					// If this exact part has not yet been actuated, an edge behind the
					// final array of the still-airborne previous part is its duplicate,
					// not permission to advance the next queue sequence.
					IF BatchSensorOrderInvalid
						AND NOT BatchCanResyncSkippedSensors
						AND (BatchNextSensorSequence[BatchLoopIndex] > 1) THEN
						BatchPreviousSlotIndex := UDINT_TO_INT(
							(BatchNextSensorSequence[BatchLoopIndex] - 2) MOD 128);
						IF (BatchQueueArrayMask[BatchPreviousSlotIndex] AND BYTE#8) <> BYTE#0 THEN
							BatchPreviousLastRequiredSensor := 8;
							BatchPreviousLastRequiredArrayMask := BYTE#8;
						ELSIF (BatchQueueArrayMask[BatchPreviousSlotIndex] AND BYTE#4) <> BYTE#0 THEN
							BatchPreviousLastRequiredSensor := 6;
							BatchPreviousLastRequiredArrayMask := BYTE#4;
						ELSIF (BatchQueueArrayMask[BatchPreviousSlotIndex] AND BYTE#2) <> BYTE#0 THEN
							BatchPreviousLastRequiredSensor := 4;
							BatchPreviousLastRequiredArrayMask := BYTE#2;
						ELSIF (BatchQueueArrayMask[BatchPreviousSlotIndex] AND BYTE#1) <> BYTE#0 THEN
							BatchPreviousLastRequiredSensor := 2;
							BatchPreviousLastRequiredArrayMask := BYTE#1;
						END_IF
						BatchIgnoreAirborneDuplicate :=
							(BatchQueueSequence[BatchPreviousSlotIndex]
								= (BatchNextSensorSequence[BatchLoopIndex] - 1))
							AND NOT BatchQueueExitSeen[BatchPreviousSlotIndex]
							AND (BatchPreviousLastRequiredArrayMask <> BYTE#0)
							AND ((BatchQueueActuatedMask[BatchPreviousSlotIndex]
								AND BatchPreviousLastRequiredArrayMask) <> BYTE#0)
							AND (BatchLoopIndex > BatchPreviousLastRequiredSensor);
					END_IF
				END_IF
				ReorientationFaultQueueSlotSequence := BatchQueueSequence[BatchSlotIndex];
				IF (BatchNextSensorSequence[BatchLoopIndex] > ReorientationQueueEnqueueAck)
					OR (BatchQueueSequence[BatchSlotIndex] <> BatchNextSensorSequence[BatchLoopIndex]) THEN
					ReorientationFaultDetail := 2;
					ReorientationWarningCode := 4;
					ReorientationWarningSensor := INT_TO_UINT(BatchLoopIndex);
					ReorientationWarningSequence := BatchNextSensorSequence[BatchLoopIndex];
					ReorientationWarningPreviousSequence := ReorientationFaultPreviousSequence;
					ReorientationWarningSkippedBarrierMask := BYTE#0;
					ReorientationWarningCounter := ReorientationWarningCounter + 1;
					IF (BatchLoopIndex MOD 2) = 1 THEN
						BatchJobIndex := (BatchLoopIndex + 1) / 2;
						PairedFirstBarrierLocked[BatchJobIndex] := TRUE;
						PairedFirstBarrierLockStartMs[BatchJobIndex] := LightBarrierEventClockMs;
						PairedSecondBarrierLocked[BatchJobIndex] := FALSE;
					ELSE
						BatchJobIndex := BatchLoopIndex / 2;
						PairedSecondBarrierLocked[BatchJobIndex] := TRUE;
						PairedSecondBarrierLockStartMs[BatchJobIndex] := LightBarrierEventClockMs;
						PairedFirstBarrierLocked[BatchJobIndex] := FALSE;
					END_IF
				ELSIF BatchIgnoreAirborneDuplicate THEN
					// The partner gate admitted another optical edge from the already
					// actuated previous part. Keep the current cursor unchanged and
					// restart this sensor's inhibit instead of faulting or misassigning it.
					ReorientationWarningCode := 2;
					ReorientationWarningSensor := INT_TO_UINT(BatchLoopIndex);
					ReorientationWarningSequence := BatchNextSensorSequence[BatchLoopIndex];
					ReorientationWarningPreviousSequence :=
						BatchNextSensorSequence[BatchLoopIndex] - 1;
					ReorientationWarningSkippedBarrierMask := BYTE#0;
					ReorientationWarningCounter := ReorientationWarningCounter + 1;
					IF (BatchLoopIndex MOD 2) = 1 THEN
						BatchJobIndex := (BatchLoopIndex + 1) / 2;
						PairedFirstBarrierLocked[BatchJobIndex] := TRUE;
						PairedFirstBarrierLockStartMs[BatchJobIndex] := LightBarrierEventClockMs;
						PairedSecondBarrierLocked[BatchJobIndex] := FALSE;
					ELSE
						BatchJobIndex := BatchLoopIndex / 2;
						PairedSecondBarrierLocked[BatchJobIndex] := TRUE;
						PairedSecondBarrierLockStartMs[BatchJobIndex] := LightBarrierEventClockMs;
						PairedFirstBarrierLocked[BatchJobIndex] := FALSE;
					END_IF
				ELSIF BatchSensorOrderInvalid AND NOT BatchCanResyncSkippedSensors THEN
					ReorientationFaultDetail := 3;
					ReorientationWarningCode := 5;
					ReorientationWarningSensor := INT_TO_UINT(BatchLoopIndex);
					ReorientationWarningSequence := BatchNextSensorSequence[BatchLoopIndex];
					ReorientationWarningPreviousSequence := ReorientationFaultPreviousSequence;
					ReorientationWarningSkippedBarrierMask := BYTE#0;
					ReorientationWarningCounter := ReorientationWarningCounter + 1;
					IF (BatchLoopIndex MOD 2) = 1 THEN
						BatchJobIndex := (BatchLoopIndex + 1) / 2;
						PairedFirstBarrierLocked[BatchJobIndex] := TRUE;
						PairedFirstBarrierLockStartMs[BatchJobIndex] := LightBarrierEventClockMs;
						PairedSecondBarrierLocked[BatchJobIndex] := FALSE;
					ELSE
						BatchJobIndex := BatchLoopIndex / 2;
						PairedSecondBarrierLocked[BatchJobIndex] := TRUE;
						PairedSecondBarrierLockStartMs[BatchJobIndex] := LightBarrierEventClockMs;
						PairedFirstBarrierLocked[BatchJobIndex] := FALSE;
					END_IF
				ELSE
					IF BatchCanResyncSkippedSensors THEN
						BatchSkippedBarrierMask := BYTE#0;
						FOR BatchResyncIndex := BatchLastRequiredSensor + 1 TO BatchLoopIndex - 1 DO
							IF BatchSensorSequence[BatchResyncIndex]
								< BatchNextSensorSequence[BatchLoopIndex] THEN
								BatchSensorSequence[BatchResyncIndex] :=
									BatchNextSensorSequence[BatchLoopIndex];
								BatchNextSensorSequence[BatchResyncIndex] :=
									BatchNextSensorSequence[BatchLoopIndex] + 1;
								BatchSensorNeedsClear[BatchResyncIndex] := FALSE;
								BatchSkippedBarrierMask := BatchSkippedBarrierMask
									OR SHL(BYTE#1, BatchResyncIndex - 1);
								// Advance the alternating pair gate just as the virtual sensor
								// acceptance advances its sequence cursor.
								IF (BatchResyncIndex MOD 2) = 1 THEN
									BatchJobIndex := (BatchResyncIndex + 1) / 2;
									PairedFirstBarrierLocked[BatchJobIndex] := TRUE;
									PairedFirstBarrierLockStartMs[BatchJobIndex] := LightBarrierEventClockMs;
									PairedSecondBarrierLocked[BatchJobIndex] := FALSE;
								ELSE
									BatchJobIndex := BatchResyncIndex / 2;
									PairedSecondBarrierLocked[BatchJobIndex] := TRUE;
									PairedSecondBarrierLockStartMs[BatchJobIndex] := LightBarrierEventClockMs;
									PairedFirstBarrierLocked[BatchJobIndex] := FALSE;
								END_IF
							END_IF
						END_FOR
						// The physical current edge was evaluated before the virtual ones;
						// re-apply it last so a skipped odd sensor in the same pair cannot
						// overwrite the correct final gate phase.
						IF (BatchLoopIndex MOD 2) = 1 THEN
							BatchJobIndex := (BatchLoopIndex + 1) / 2;
							PairedFirstBarrierLocked[BatchJobIndex] := TRUE;
							PairedFirstBarrierLockStartMs[BatchJobIndex] := LightBarrierEventClockMs;
							PairedSecondBarrierLocked[BatchJobIndex] := FALSE;
						ELSE
							BatchJobIndex := BatchLoopIndex / 2;
							PairedSecondBarrierLocked[BatchJobIndex] := TRUE;
							PairedSecondBarrierLockStartMs[BatchJobIndex] := LightBarrierEventClockMs;
							PairedFirstBarrierLocked[BatchJobIndex] := FALSE;
						END_IF
						ReorientationWarningCode := 1;
						ReorientationWarningSensor := INT_TO_UINT(BatchLoopIndex);
						ReorientationWarningSequence := BatchNextSensorSequence[BatchLoopIndex];
						ReorientationWarningPreviousSequence := ReorientationFaultPreviousSequence;
						ReorientationWarningSkippedBarrierMask := BatchSkippedBarrierMask;
						ReorientationWarningCounter := ReorientationWarningCounter + 1;
					END_IF
					BatchSensorSequence[BatchLoopIndex] := BatchNextSensorSequence[BatchLoopIndex];
					IF (BatchLoopIndex MOD 2) = 1 THEN
						BatchJobIndex := (BatchLoopIndex + 1) / 2;
						BatchQueuePairStartMs[BatchSlotIndex, BatchJobIndex] := LightBarrierEventClockMs;
						IF BatchLoopIndex = 1 THEN
							ReorientationQueueEnteredCount := ReorientationQueueEnteredCount + 1;
						END_IF
					ELSE
						BatchJobIndex := BatchLoopIndex / 2;
						IF (BatchQueueArrayMask[BatchSlotIndex] AND SHL(BYTE#1, BatchJobIndex - 1)) <> BYTE#0 THEN
							IF BatchJobCount[BatchJobIndex] >= 16 THEN
								ReorientationFaultCode := 95; // per-array job FIFO overflow
								ReorientationState := 95;
								ReorientationSafeLatch := TRUE;
							ELSE
								BatchElapsedMs := LightBarrierEventClockMs - BatchQueuePairStartMs[BatchSlotIndex, BatchJobIndex];
								BatchNozzleCount := 0;
								FOR BatchSlotIndex := 0 TO 5 DO
									IF (BatchQueueNozzleMask[UDINT_TO_INT((BatchNextSensorSequence[BatchLoopIndex] - 1) MOD 128), BatchJobIndex]
										AND SHL(BYTE#1, BatchSlotIndex)) <> BYTE#0 THEN
										BatchNozzleCount := BatchNozzleCount + 1;
									END_IF
								END_FOR
								BatchSlotIndex := UDINT_TO_INT((BatchNextSensorSequence[BatchLoopIndex] - 1) MOD 128);
				// One response-delay setting is used for every nozzle count.
				BatchResponseDelayMs := BatchQueueForceSingleMs[BatchSlotIndex, BatchJobIndex];
				BatchComputedDelayMs := UINT_TO_REAL(BatchQueueDelayMs[BatchSlotIndex, BatchJobIndex]);
				IF (BatchElapsedMs > 0) AND (BatchPairSpacingMm[BatchJobIndex] > 0.0)
					AND ((BatchSensorToArraySpacingMm[BatchJobIndex]
					+ BatchQueueOffsetMm[BatchSlotIndex, BatchJobIndex]) > 0.0) THEN
					BatchComputedDelayMs := BatchComputedDelayMs
						+ (BatchSensorToArraySpacingMm[BatchJobIndex]
						+ BatchQueueOffsetMm[BatchSlotIndex, BatchJobIndex])
						* UDINT_TO_REAL(BatchElapsedMs) / BatchPairSpacingMm[BatchJobIndex]
						- BatchResponseDelayMs;
								END_IF
								IF BatchComputedDelayMs < 0.0 THEN BatchComputedDelayMs := 0.0; END_IF
								IF BatchComputedDelayMs > 31000.0 THEN BatchComputedDelayMs := 31000.0; END_IF
								BatchJobSequence[BatchJobTail[BatchJobIndex], BatchJobIndex] := BatchQueueSequence[BatchSlotIndex];
								BatchJobNozzleMask[BatchJobTail[BatchJobIndex], BatchJobIndex] := BatchQueueNozzleMask[BatchSlotIndex, BatchJobIndex];
								BatchJobPressureMbar[BatchJobTail[BatchJobIndex], BatchJobIndex] := BatchQueuePressureMbar[BatchSlotIndex, BatchJobIndex];
								BatchJobDelayCycles[BatchJobTail[BatchJobIndex], BatchJobIndex] := REAL_TO_INT(BatchComputedDelayMs);
								BatchJobPulseCycles[BatchJobTail[BatchJobIndex], BatchJobIndex] := UINT_TO_INT(BatchQueuePulseMs[BatchSlotIndex, BatchJobIndex]);
								BatchJobTail[BatchJobIndex] := (BatchJobTail[BatchJobIndex] + 1) MOD 16;
								BatchJobCount[BatchJobIndex] := BatchJobCount[BatchJobIndex] + 1;
								BatchQueueTriggeredMask[BatchSlotIndex] := BatchQueueTriggeredMask[BatchSlotIndex]
									OR SHL(BYTE#1, BatchJobIndex - 1);
							END_IF
						END_IF
						IF BatchLoopIndex = 8 THEN
							BatchQueueExitSeen[BatchSlotIndex] := TRUE;
							ReorientationExitSeen := TRUE;
						END_IF
					END_IF
					BatchNextSensorSequence[BatchLoopIndex] := BatchNextSensorSequence[BatchLoopIndex] + 1;
				END_IF
			END_IF
		END_IF
		// Preserve the first faulting sensor and its context. Without EXIT, a
		// second edge in this same 1-ms scan could overwrite the diagnostics.
		IF ReorientationSafeLatch THEN
			EXIT;
		END_IF
	END_FOR
END_IF

ReorientationSensorSequence1 := BatchSensorSequence[1];
ReorientationSensorSequence2 := BatchSensorSequence[2];
ReorientationSensorSequence3 := BatchSensorSequence[3];
ReorientationSensorSequence4 := BatchSensorSequence[4];
ReorientationSensorSequence5 := BatchSensorSequence[5];
ReorientationSensorSequence6 := BatchSensorSequence[6];
ReorientationSensorSequence7 := BatchSensorSequence[7];
ReorientationSensorSequence8 := BatchSensorSequence[8];

// Accept either signal polarity, but only after the new state remains stable for the debounce time.
// The candidate position is captured on the first cycle of the ultimately stable transition.
IF BarrierCalibrationActive THEN
	IF NOT BarrierCalibrationFirstCaptured THEN
		IF BarrierCalibrationFirstState <> BarrierCalibrationFirstInitialState THEN
			IF BarrierCalibrationFirstStableCycles = 0 THEN
				BarrierCalibrationFirstCandidatePosition := StepperInternalPosition;
			END_IF
			IF BarrierCalibrationFirstStableCycles < GuiBarrierCalibrationDebounceMs THEN
				BarrierCalibrationFirstStableCycles := BarrierCalibrationFirstStableCycles + 1;
			END_IF
			IF BarrierCalibrationFirstStableCycles >= GuiBarrierCalibrationDebounceMs THEN
				BarrierCalibrationFirstPosition := BarrierCalibrationFirstCandidatePosition;
				BarrierCalibrationFirstCaptured := TRUE;
				BarrierCalibrationStatusCode := 2;
			END_IF
		ELSE
			BarrierCalibrationFirstStableCycles := 0;
		END_IF
	ELSIF BarrierCalibrationFirstCaptured
		AND NOT BarrierCalibrationSecondCaptured THEN
		IF BarrierCalibrationSecondState <> BarrierCalibrationSecondInitialState THEN
			IF BarrierCalibrationSecondStableCycles = 0 THEN
				BarrierCalibrationSecondCandidatePosition := StepperInternalPosition;
			END_IF
			IF BarrierCalibrationSecondStableCycles < GuiBarrierCalibrationDebounceMs THEN
				BarrierCalibrationSecondStableCycles := BarrierCalibrationSecondStableCycles + 1;
			END_IF
			IF BarrierCalibrationSecondStableCycles >= GuiBarrierCalibrationDebounceMs THEN
				BarrierCalibrationSecondPosition := BarrierCalibrationSecondCandidatePosition;
				BarrierCalibrationSecondCaptured := TRUE;
				BarrierCalibrationPositionDelta := UDINT_TO_LINT(BarrierCalibrationSecondPosition)
					- UDINT_TO_LINT(BarrierCalibrationFirstPosition);
				IF BarrierCalibrationPositionDelta > LINT#2147483647 THEN
					BarrierCalibrationPositionDelta := BarrierCalibrationPositionDelta - LINT#4294967296;
				ELSIF BarrierCalibrationPositionDelta < LINT#-2147483648 THEN
					BarrierCalibrationPositionDelta := BarrierCalibrationPositionDelta + LINT#4294967296;
				END_IF
				IF BarrierCalibrationPositionDelta < 0 THEN
					BarrierCalibrationPositionDelta := -BarrierCalibrationPositionDelta;
				END_IF
				IF BarrierCalibrationPositionDelta > 0 THEN
					BarrierCalibrationDifferenceIncrements := LINT_TO_UDINT(BarrierCalibrationPositionDelta);
					BarrierCalibrationDistanceMm :=
						TO_REAL(BarrierCalibrationDifferenceIncrements) / 64.0 * GuiConveyorMmPerFullStep;
					BarrierCalibrationValid := TRUE;
					BarrierCalibrationStatusCode := 3;
				ELSE
					BarrierCalibrationDifferenceIncrements := 0;
					BarrierCalibrationDistanceMm := 0.0;
					BarrierCalibrationValid := FALSE;
					BarrierCalibrationStatusCode := 4;
				END_IF
				BarrierCalibrationActive := FALSE;
				GuiCalibrationStop := TRUE;
			END_IF
		ELSE
			BarrierCalibrationSecondStableCycles := 0;
		END_IF
	END_IF
END_IF

// Cancel a measurement if the drive stops before the second selected barrier is reached.
IF BarrierCalibrationActive
	AND (BarrierCalibrationAbortRequested
		OR ((ConveyorMotionState = 0) AND (ConveyorMotionMode = 0))) THEN
	BarrierCalibrationActive := FALSE;
	BarrierCalibrationValid := FALSE;
	IF StepperPosError THEN
		BarrierCalibrationStatusCode := 5;
	ELSE
		BarrierCalibrationStatusCode := 4;
	END_IF
END_IF

IF NOT GuiReorientationControlActive AND PairedSecondBarrierFalling[1] AND Array1Active AND (State <= 2) THEN
	Array1TriggerPending := TRUE;
END_IF

IF NOT GuiReorientationControlActive AND PairedSecondBarrierFalling[2] AND Array2Active AND (State2 = 2) THEN
	Array2TriggerPending := TRUE;
END_IF

IF NOT GuiReorientationControlActive AND PairedSecondBarrierFalling[3] AND Array3Active AND (State3 <= 2) THEN
	Array3TriggerPending := TRUE;
END_IF

IF NOT GuiReorientationControlActive AND PairedSecondBarrierFalling[4] AND Array4Active AND (State4 = 2) THEN
	Array4TriggerPending := TRUE;
END_IF

// Measure the selected force-sensor peak relative to a debounced light-barrier edge.
IF GuiForceDelayLightBarrier = 2 THEN
	ForceDelayTrigger := PairedSecondBarrierFalling[1];
ELSIF GuiForceDelayLightBarrier = 4 THEN
	ForceDelayTrigger := PairedSecondBarrierFalling[2];
ELSIF GuiForceDelayLightBarrier = 6 THEN
	ForceDelayTrigger := PairedSecondBarrierFalling[3];
ELSE
	ForceDelayTrigger := PairedSecondBarrierFalling[4];
END_IF

IF GuiForceDelaySensor = 2 THEN
	ForceDelayCurrentSignal := NozzlePressure2;
ELSE
	ForceDelayCurrentSignal := NozzlePressure;
END_IF

IF GuiForceDelayReset THEN
	ForceDelayBusy := FALSE;
	ForceDelayResultCounter := 0;
	ForceDelayValidCount := 0;
	ForceDelayInvalidCount := 0;
	ForceDelayLastValid := FALSE;
	ForceDelayLightBarrierTimeMs := 0;
	ForceDelayPeakTimeMs := 0;
	ForceDelayPeakDelayMs := 0;
	ForceDelayElapsedMs := 0;
	ForceDelayBaseline := 0.0;
	ForceDelayPeak := 0.0;
	ForceDelayPeakRise := 0.0;
	GuiForceDelayReset := FALSE;
END_IF

IF NOT GuiForceDelayMeasurementEnabled THEN
	ForceDelayBusy := FALSE;
	ForceDelayStatusCode := 0;
ELSE
	IF GuiForceDelayWindowMs < 100 THEN
		GuiForceDelayWindowMs := 100;
	ELSIF GuiForceDelayWindowMs > 30000 THEN
		GuiForceDelayWindowMs := 30000;
	END_IF
	IF GuiForceDelayMinRise < 0.0 THEN
		GuiForceDelayMinRise := 0.0;
	END_IF

	IF ForceDelayBusy THEN
		IF ForceDelayElapsedMs < 30000 THEN
			ForceDelayElapsedMs := ForceDelayElapsedMs + 1;
		END_IF
		IF ForceDelayCurrentSignal > ForceDelayPeak THEN
			ForceDelayPeak := ForceDelayCurrentSignal;
			ForceDelayPeakDelayMs := UINT_TO_UDINT(ForceDelayElapsedMs);
		END_IF
		IF ForceDelayElapsedMs >= GuiForceDelayWindowMs THEN
			ForceDelayPeakRise := ForceDelayPeak - ForceDelayBaseline;
			ForceDelayPeakTimeMs := ForceDelayLightBarrierTimeMs + ForceDelayPeakDelayMs;
			ForceDelayLastValid := ForceDelayPeakRise >= GuiForceDelayMinRise;
			ForceDelayResultCounter := ForceDelayResultCounter + 1;
			IF ForceDelayLastValid THEN
				ForceDelayValidCount := ForceDelayValidCount + 1;
				ForceDelayStatusCode := 3;
			ELSE
				ForceDelayInvalidCount := ForceDelayInvalidCount + 1;
				ForceDelayStatusCode := 4;
			END_IF
			ForceDelayBusy := FALSE;
		END_IF
	ELSIF ForceDelayTrigger THEN
		IF ForceDelayBaselineCount > 0 THEN
			IF GuiForceDelaySensor = 2 THEN
				ForceDelayBaseline := ForceDelayBaselineSum2 / UINT_TO_REAL(ForceDelayBaselineCount);
			ELSE
				ForceDelayBaseline := ForceDelayBaselineSum1 / UINT_TO_REAL(ForceDelayBaselineCount);
			END_IF
		ELSE
			ForceDelayBaseline := ForceDelayCurrentSignal;
		END_IF
		ForceDelayLightBarrierTimeMs := LightBarrierEventClockMs;
		ForceDelayPeak := ForceDelayCurrentSignal;
		ForceDelayPeakRise := 0.0;
		ForceDelayPeakDelayMs := 0;
		ForceDelayElapsedMs := 0;
		ForceDelayBusy := TRUE;
		ForceDelayStatusCode := 2;
	ELSIF (ForceDelayStatusCode = 0) OR (ForceDelayStatusCode = 2) THEN
		ForceDelayStatusCode := 1;
	END_IF
END_IF

// Keep a 50 ms pre-trigger baseline for both analogue channels.
IF NOT ForceDelayBusy THEN
	ForceDelayBaselineSum1 := ForceDelayBaselineSum1 - ForceDelayBaselineBuffer1[ForceDelayBaselineIndex];
	ForceDelayBaselineSum2 := ForceDelayBaselineSum2 - ForceDelayBaselineBuffer2[ForceDelayBaselineIndex];
	ForceDelayBaselineBuffer1[ForceDelayBaselineIndex] := NozzlePressure;
	ForceDelayBaselineBuffer2[ForceDelayBaselineIndex] := NozzlePressure2;
	ForceDelayBaselineSum1 := ForceDelayBaselineSum1 + NozzlePressure;
	ForceDelayBaselineSum2 := ForceDelayBaselineSum2 + NozzlePressure2;
	IF ForceDelayBaselineCount < 50 THEN
		ForceDelayBaselineCount := ForceDelayBaselineCount + 1;
	END_IF
	IF ForceDelayBaselineIndex >= 49 THEN
		ForceDelayBaselineIndex := 0;
	ELSE
		ForceDelayBaselineIndex := ForceDelayBaselineIndex + 1;
	END_IF
END_IF

// Falling edge on light barrier 1 starts the velocity timing window.
IF PairedFirstBarrierFalling[1] THEN
	VelocityTimingActive := FALSE;
	VelocityTimer(IN := FALSE, PT := T#30S);
	VelocityTimingActive := TRUE;
	VelocityMeasurementValid := FALSE;
	EstimatedVelocityMmPerSec := 0.0;
	EstimatedVelocityMmPerSec1 := 0.0;
	EstimatedOffsetDelayMs1 := 0.0;
	OffsetDelayCycles1 := 0;
END_IF

// Light barriers 1 and 2 measure velocity for nozzle array 1.
// Light barrier 2 is also the physical trigger for nozzle array 1.
IF PairedSecondBarrierFalling[1] THEN
	IF VelocityTimingActive AND (TIME_TO_INT(VelocityTimer.ET) > 0) AND (GuiSensorSpacing12Mm > 0.0) THEN
		LastVelocityTimeMs := TIME_TO_INT(VelocityTimer.ET);
		EstimatedVelocityMmPerSec := GuiSensorSpacing12Mm * 1000.0 / TO_REAL(LastVelocityTimeMs);
		EstimatedVelocityMmPerSec1 := EstimatedVelocityMmPerSec;
		VelocityMeasurementValid := TRUE;
	END_IF
	VelocityTimingActive := FALSE;
END_IF

// Light barriers 3 and 4 measure velocity for nozzle array 2.
IF PairedFirstBarrierFalling[2] THEN
	VelocityTiming2Active := FALSE;
	VelocityTimer2(IN := FALSE, PT := T#30S);
	VelocityTiming2Active := TRUE;
	VelocityMeasurement2Valid := FALSE;
	EstimatedVelocityMmPerSec2 := 0.0;
	EstimatedOffsetDelayMs2 := 0.0;
	OffsetDelayCycles2 := 0;
END_IF

// Light barrier 4 completes the array 2 velocity measurement and triggers array 2.
IF PairedSecondBarrierFalling[2] THEN
	IF VelocityTiming2Active AND (TIME_TO_INT(VelocityTimer2.ET) > 0) AND (GuiSensorSpacing34Mm > 0.0) THEN
		LastVelocityTime2Ms := TIME_TO_INT(VelocityTimer2.ET);
		EstimatedVelocityMmPerSec2 := GuiSensorSpacing34Mm * 1000.0 / TO_REAL(LastVelocityTime2Ms);
		VelocityMeasurement2Valid := TRUE;
	END_IF
	VelocityTiming2Active := FALSE;
END_IF

// Light barriers 5 and 6 measure velocity for nozzle array 3.
IF PairedFirstBarrierFalling[3] THEN
	VelocityTiming3Active := FALSE;
	VelocityTimer3(IN := FALSE, PT := T#30S);
	VelocityTiming3Active := TRUE;
	VelocityMeasurement3Valid := FALSE;
	EstimatedVelocityMmPerSec3 := 0.0;
	EstimatedOffsetDelayMs3 := 0.0;
	OffsetDelayCycles3 := 0;
END_IF

// Light barrier 6 completes the array 3 velocity measurement and triggers array 3.
IF PairedSecondBarrierFalling[3] THEN
	IF VelocityTiming3Active AND (TIME_TO_INT(VelocityTimer3.ET) > 0) AND (GuiSensorSpacing56Mm > 0.0) THEN
		LastVelocityTime3Ms := TIME_TO_INT(VelocityTimer3.ET);
		EstimatedVelocityMmPerSec3 := GuiSensorSpacing56Mm * 1000.0 / TO_REAL(LastVelocityTime3Ms);
		VelocityMeasurement3Valid := TRUE;
	END_IF
	VelocityTiming3Active := FALSE;
END_IF

// Light barriers 7 and 8 measure velocity for nozzle array 4.
IF PairedFirstBarrierFalling[4] THEN
	VelocityTiming4Active := FALSE;
	VelocityTimer4(IN := FALSE, PT := T#30S);
	VelocityTiming4Active := TRUE;
	VelocityMeasurement4Valid := FALSE;
	EstimatedVelocityMmPerSec4 := 0.0;
	EstimatedOffsetDelayMs4 := 0.0;
	OffsetDelayCycles4 := 0;
END_IF

// Light barrier 8 completes the array 4 velocity measurement and triggers array 4.
IF PairedSecondBarrierFalling[4] THEN
	IF VelocityTiming4Active AND (TIME_TO_INT(VelocityTimer4.ET) > 0) AND (GuiSensorSpacing78Mm > 0.0) THEN
		LastVelocityTime4Ms := TIME_TO_INT(VelocityTimer4.ET);
		EstimatedVelocityMmPerSec4 := GuiSensorSpacing78Mm * 1000.0 / TO_REAL(LastVelocityTime4Ms);
		VelocityMeasurement4Valid := TRUE;
	END_IF
	VelocityTiming4Active := FALSE;
END_IF

IF GuiPressureMbar1 < 0 THEN
	PresValueV02 := 0;
ELSIF GuiPressureMbar1 > 6000 THEN
	PresValueV02 := 6000;
ELSE
	PresValueV02 := GuiPressureMbar1;
END_IF

IF GuiPressureMbar2 < 0 THEN
	PresValueV04 := 0;
ELSIF GuiPressureMbar2 > 6000 THEN
	PresValueV04 := 6000;
ELSE
	PresValueV04 := GuiPressureMbar2;
END_IF

IF GuiPressureMbar3 < 0 THEN
	PresValueV12 := 0;
ELSIF GuiPressureMbar3 > 6000 THEN
	PresValueV12 := 6000;
ELSE
	PresValueV12 := GuiPressureMbar3;
END_IF

IF GuiPressureMbar4 < 0 THEN
	PresValueV14 := 0;
ELSIF GuiPressureMbar4 > 6000 THEN
	PresValueV14 := 6000;
ELSE
	PresValueV14 := GuiPressureMbar4;
END_IF

IF GuiPulseDurationMs1 < 1 THEN
	ShotDurationCycles := 1;
ELSIF GuiPulseDurationMs1 > 500 THEN
	ShotDurationCycles := 500;
ELSE
	ShotDurationCycles := UINT_TO_INT(GuiPulseDurationMs1);
END_IF

IF GuiPulseDurationMs2 < 1 THEN
	ShotDurationCycles2 := 1;
ELSIF GuiPulseDurationMs2 > 500 THEN
	ShotDurationCycles2 := 500;
ELSE
	ShotDurationCycles2 := UINT_TO_INT(GuiPulseDurationMs2);
END_IF

IF GuiPulseDurationMs3 < 1 THEN
	ShotDurationCycles3 := 1;
ELSIF GuiPulseDurationMs3 > 500 THEN
	ShotDurationCycles3 := 500;
ELSE
	ShotDurationCycles3 := UINT_TO_INT(GuiPulseDurationMs3);
END_IF

IF GuiPulseDurationMs4 < 1 THEN
	ShotDurationCycles4 := 1;
ELSIF GuiPulseDurationMs4 > 500 THEN
	ShotDurationCycles4 := 500;
ELSE
	ShotDurationCycles4 := UINT_TO_INT(GuiPulseDurationMs4);
END_IF

IF GuiDelayMs1 > 1000 THEN
	DelayDurationCycles := 1000;
ELSE
	DelayDurationCycles := UINT_TO_INT(GuiDelayMs1);
END_IF

IF GuiDelayMs2 > 1000 THEN
	DelayDurationCycles2 := 1000;
ELSE
	DelayDurationCycles2 := UINT_TO_INT(GuiDelayMs2);
END_IF

IF GuiDelayMs3 > 1000 THEN
	DelayDurationCycles3 := 1000;
ELSE
	DelayDurationCycles3 := UINT_TO_INT(GuiDelayMs3);
END_IF

IF GuiDelayMs4 > 1000 THEN
	DelayDurationCycles4 := 1000;
ELSE
	DelayDurationCycles4 := UINT_TO_INT(GuiDelayMs4);
END_IF

IF GuiForceResponseDelayMs1 < 0.0 THEN
	GuiForceResponseDelayMs1 := 0.0;
ELSIF GuiForceResponseDelayMs1 > 1000.0 THEN
	GuiForceResponseDelayMs1 := 1000.0;
END_IF
IF GuiForceResponseDelayMs2 < 0.0 THEN
	GuiForceResponseDelayMs2 := 0.0;
ELSIF GuiForceResponseDelayMs2 > 1000.0 THEN
	GuiForceResponseDelayMs2 := 1000.0;
END_IF
IF GuiForceResponseDelayMs3 < 0.0 THEN
	GuiForceResponseDelayMs3 := 0.0;
ELSIF GuiForceResponseDelayMs3 > 1000.0 THEN
	GuiForceResponseDelayMs3 := 1000.0;
END_IF
IF GuiForceResponseDelayMs4 < 0.0 THEN
	GuiForceResponseDelayMs4 := 0.0;
ELSIF GuiForceResponseDelayMs4 > 1000.0 THEN
	GuiForceResponseDelayMs4 := 1000.0;
END_IF

IF GuiForceSingleNozzleResponseDelayMs1 < 0.0 THEN
	GuiForceSingleNozzleResponseDelayMs1 := 0.0;
ELSIF GuiForceSingleNozzleResponseDelayMs1 > 1000.0 THEN
	GuiForceSingleNozzleResponseDelayMs1 := 1000.0;
END_IF
IF GuiForceSingleNozzleResponseDelayMs2 < 0.0 THEN
	GuiForceSingleNozzleResponseDelayMs2 := 0.0;
ELSIF GuiForceSingleNozzleResponseDelayMs2 > 1000.0 THEN
	GuiForceSingleNozzleResponseDelayMs2 := 1000.0;
END_IF
IF GuiForceSingleNozzleResponseDelayMs3 < 0.0 THEN
	GuiForceSingleNozzleResponseDelayMs3 := 0.0;
ELSIF GuiForceSingleNozzleResponseDelayMs3 > 1000.0 THEN
	GuiForceSingleNozzleResponseDelayMs3 := 1000.0;
END_IF
IF GuiForceSingleNozzleResponseDelayMs4 < 0.0 THEN
	GuiForceSingleNozzleResponseDelayMs4 := 0.0;
ELSIF GuiForceSingleNozzleResponseDelayMs4 > 1000.0 THEN
	GuiForceSingleNozzleResponseDelayMs4 := 1000.0;
END_IF

// Interpolate the measured response delay from one to four enabled nozzles.
ActiveNozzleCount1 := 0;
IF GuiNozzleEnabled1 THEN ActiveNozzleCount1 := ActiveNozzleCount1 + 1; END_IF
IF GuiNozzleEnabled2 THEN ActiveNozzleCount1 := ActiveNozzleCount1 + 1; END_IF
IF GuiNozzleEnabled3 THEN ActiveNozzleCount1 := ActiveNozzleCount1 + 1; END_IF
IF GuiNozzleEnabled4 THEN ActiveNozzleCount1 := ActiveNozzleCount1 + 1; END_IF
IF GuiNozzleEnabled5 THEN ActiveNozzleCount1 := ActiveNozzleCount1 + 1; END_IF
IF GuiNozzleEnabled6 THEN ActiveNozzleCount1 := ActiveNozzleCount1 + 1; END_IF
ActiveNozzleCount2 := 0;
IF GuiNozzleEnabled7 THEN ActiveNozzleCount2 := ActiveNozzleCount2 + 1; END_IF
IF GuiNozzleEnabled8 THEN ActiveNozzleCount2 := ActiveNozzleCount2 + 1; END_IF
IF GuiNozzleEnabled9 THEN ActiveNozzleCount2 := ActiveNozzleCount2 + 1; END_IF
IF GuiNozzleEnabled10 THEN ActiveNozzleCount2 := ActiveNozzleCount2 + 1; END_IF
IF GuiNozzleEnabled11 THEN ActiveNozzleCount2 := ActiveNozzleCount2 + 1; END_IF
IF GuiNozzleEnabled12 THEN ActiveNozzleCount2 := ActiveNozzleCount2 + 1; END_IF
ActiveNozzleCount3 := 0;
IF GuiNozzleEnabled13 THEN ActiveNozzleCount3 := ActiveNozzleCount3 + 1; END_IF
IF GuiNozzleEnabled14 THEN ActiveNozzleCount3 := ActiveNozzleCount3 + 1; END_IF
IF GuiNozzleEnabled15 THEN ActiveNozzleCount3 := ActiveNozzleCount3 + 1; END_IF
IF GuiNozzleEnabled16 THEN ActiveNozzleCount3 := ActiveNozzleCount3 + 1; END_IF
IF GuiNozzleEnabled17 THEN ActiveNozzleCount3 := ActiveNozzleCount3 + 1; END_IF
IF GuiNozzleEnabled18 THEN ActiveNozzleCount3 := ActiveNozzleCount3 + 1; END_IF
ActiveNozzleCount4 := 0;
IF GuiNozzleEnabled19 THEN ActiveNozzleCount4 := ActiveNozzleCount4 + 1; END_IF
IF GuiNozzleEnabled20 THEN ActiveNozzleCount4 := ActiveNozzleCount4 + 1; END_IF
IF GuiNozzleEnabled21 THEN ActiveNozzleCount4 := ActiveNozzleCount4 + 1; END_IF
IF GuiNozzleEnabled22 THEN ActiveNozzleCount4 := ActiveNozzleCount4 + 1; END_IF
IF GuiNozzleEnabled23 THEN ActiveNozzleCount4 := ActiveNozzleCount4 + 1; END_IF
IF GuiNozzleEnabled24 THEN ActiveNozzleCount4 := ActiveNozzleCount4 + 1; END_IF

// The legacy four-nozzle variables remain in the ADS interface, but the same
// single force-response value is now used for every active-nozzle count.
EffectiveForceResponseDelayMs1 := GuiForceSingleNozzleResponseDelayMs1;
EffectiveForceResponseDelayMs2 := GuiForceSingleNozzleResponseDelayMs2;
EffectiveForceResponseDelayMs3 := GuiForceSingleNozzleResponseDelayMs3;
EffectiveForceResponseDelayMs4 := GuiForceSingleNozzleResponseDelayMs4;

IF NOT GuiReorientationControlActive AND VelocityMeasurementValid AND (EstimatedVelocityMmPerSec1 > 0.0) THEN
	IF (GuiSensor2ToArray1SpacingMm + GuiOffsetMm1) <= 0.0 THEN
		EstimatedOffsetDelayMs1 := 0.0;
	ELSE
		EstimatedOffsetDelayMs1 := ((GuiSensor2ToArray1SpacingMm + GuiOffsetMm1)
			* 1000.0 / EstimatedVelocityMmPerSec1) - EffectiveForceResponseDelayMs1;
		IF EstimatedOffsetDelayMs1 < 0.0 THEN
			EstimatedOffsetDelayMs1 := 0.0;
		END_IF
	END_IF
ELSE
	EstimatedOffsetDelayMs1 := 0.0;
END_IF

IF NOT GuiReorientationControlActive AND VelocityMeasurement2Valid AND (EstimatedVelocityMmPerSec2 > 0.0) THEN
	IF (GuiSensor4ToArray2SpacingMm + GuiOffsetMm2) <= 0.0 THEN
		EstimatedOffsetDelayMs2 := 0.0;
	ELSE
		EstimatedOffsetDelayMs2 := ((GuiSensor4ToArray2SpacingMm + GuiOffsetMm2)
			* 1000.0 / EstimatedVelocityMmPerSec2) - EffectiveForceResponseDelayMs2;
		IF EstimatedOffsetDelayMs2 < 0.0 THEN
			EstimatedOffsetDelayMs2 := 0.0;
		END_IF
	END_IF
ELSE
	EstimatedOffsetDelayMs2 := 0.0;
END_IF

IF NOT GuiReorientationControlActive AND VelocityMeasurement3Valid AND (EstimatedVelocityMmPerSec3 > 0.0) THEN
	IF (GuiSensor6ToArray3SpacingMm + GuiOffsetMm3) <= 0.0 THEN
		EstimatedOffsetDelayMs3 := 0.0;
	ELSE
		EstimatedOffsetDelayMs3 := ((GuiSensor6ToArray3SpacingMm + GuiOffsetMm3)
			* 1000.0 / EstimatedVelocityMmPerSec3) - EffectiveForceResponseDelayMs3;
		IF EstimatedOffsetDelayMs3 < 0.0 THEN
			EstimatedOffsetDelayMs3 := 0.0;
		END_IF
	END_IF
ELSE
	EstimatedOffsetDelayMs3 := 0.0;
END_IF

IF NOT GuiReorientationControlActive AND VelocityMeasurement4Valid AND (EstimatedVelocityMmPerSec4 > 0.0) THEN
	IF (GuiSensor8ToArray4SpacingMm + GuiOffsetMm4) <= 0.0 THEN
		EstimatedOffsetDelayMs4 := 0.0;
	ELSE
		EstimatedOffsetDelayMs4 := ((GuiSensor8ToArray4SpacingMm + GuiOffsetMm4)
			* 1000.0 / EstimatedVelocityMmPerSec4) - EffectiveForceResponseDelayMs4;
		IF EstimatedOffsetDelayMs4 < 0.0 THEN
			EstimatedOffsetDelayMs4 := 0.0;
		END_IF
	END_IF
ELSE
	EstimatedOffsetDelayMs4 := 0.0;
END_IF

IF EstimatedOffsetDelayMs1 > 30000.0 THEN
	OffsetDelayCycles1 := 30000;
ELSE
	OffsetDelayCycles1 := REAL_TO_INT(EstimatedOffsetDelayMs1);
END_IF

IF EstimatedOffsetDelayMs2 > 30000.0 THEN
	OffsetDelayCycles2 := 30000;
ELSE
	OffsetDelayCycles2 := REAL_TO_INT(EstimatedOffsetDelayMs2);
END_IF

IF EstimatedOffsetDelayMs3 > 30000.0 THEN
	OffsetDelayCycles3 := 30000;
ELSE
	OffsetDelayCycles3 := REAL_TO_INT(EstimatedOffsetDelayMs3);
END_IF

IF EstimatedOffsetDelayMs4 > 30000.0 THEN
	OffsetDelayCycles4 := 30000;
ELSE
	OffsetDelayCycles4 := REAL_TO_INT(EstimatedOffsetDelayMs4);
END_IF

DelayDurationCycles := DelayDurationCycles + OffsetDelayCycles1;
DelayDurationCycles2 := DelayDurationCycles2 + OffsetDelayCycles2;
DelayDurationCycles3 := DelayDurationCycles3 + OffsetDelayCycles3;
DelayDurationCycles4 := DelayDurationCycles4 + OffsetDelayCycles4;

CASE State OF
	0:
		Enable0 := TRUE;
		Acknowledge0 := FALSE;
		State := State + 1;
		
	1:
		Enable0 := TRUE;
		Acknowledge0 := TRUE;
		State := State + 1;
	2:
		//start nozzle array 1 on the falling edge of light barrier 2
		IF NOT Array1Active THEN
			Array1TriggerPending := FALSE;
		ELSIF Array1TriggerPending THEN
			Array1TriggerPending := FALSE;
			Counter := 0;
			LatchedDelayCycles1 := DelayDurationCycles;
			LatchedNozzleEndCycles1 := DelayDurationCycles + ShotDurationCycles;
			PressureSum := 0.0;
			PressureSum1 := 0.0;
			PressureSum2 := 0.0;
			PressurePoints := 0;
			PressurePoints1 := 0;
			PressurePoints2 := 0;
			State := State + 1;
		END_IF
	3:
		IF NOT Array1Active THEN
			OpenValve1 := FALSE;
			OpenValve2 := FALSE;
			OpenValve3 := FALSE;
			OpenValve4 := FALSE;
			OpenValve17 := FALSE;
			OpenValve18 := FALSE;
			Counter := 0;
			State := 2;
		ELSE
			Counter := Counter + 1;
			OpenValve1 := GuiArrayEnabled1 AND GuiNozzleEnabled1 AND (Counter > LatchedDelayCycles1) AND (Counter <= LatchedNozzleEndCycles1);
			OpenValve2 := GuiArrayEnabled1 AND GuiNozzleEnabled2 AND (Counter > LatchedDelayCycles1) AND (Counter <= LatchedNozzleEndCycles1);
			OpenValve3 := GuiArrayEnabled1 AND GuiNozzleEnabled3 AND (Counter > LatchedDelayCycles1) AND (Counter <= LatchedNozzleEndCycles1);
			OpenValve4 := GuiArrayEnabled1 AND GuiNozzleEnabled4 AND (Counter > LatchedDelayCycles1) AND (Counter <= LatchedNozzleEndCycles1);
			OpenValve17 := GuiArrayEnabled1 AND GuiNozzleEnabled5 AND (Counter > LatchedDelayCycles1) AND (Counter <= LatchedNozzleEndCycles1);
			OpenValve18 := GuiArrayEnabled1 AND GuiNozzleEnabled6 AND (Counter > LatchedDelayCycles1) AND (Counter <= LatchedNozzleEndCycles1);
			IF GuiReorientationControlActive AND (BatchActiveSequence[1] > 0)
				AND (OpenValve1 OR OpenValve2 OR OpenValve3 OR OpenValve4 OR OpenValve17 OR OpenValve18) THEN
				BatchSlotIndex := UDINT_TO_INT((BatchActiveSequence[1] - 1) MOD 128);
				BatchQueueActuatedMask[BatchSlotIndex] := BatchQueueActuatedMask[BatchSlotIndex] OR BYTE#1;
			END_IF

			IF OpenValve1 OR OpenValve2 OR OpenValve3 OR OpenValve4 OR OpenValve17 OR OpenValve18 THEN
				PressureSum := PressureSum + NozzlePressure;
				PressureSum1 := PressureSum1 + NozzlePressure;
				PressurePoints := PressurePoints + 1;
				PressurePoints1 := PressurePoints1 + 1;
				IF PressurePoints1 <= 1000 THEN
					N1PressureValues[PressurePoints1] := NozzlePressure;
				END_IF
				PressureSum := PressureSum + NozzlePressure2;
				PressureSum2 := PressureSum2 + NozzlePressure2;
				PressurePoints := PressurePoints + 1;
				PressurePoints2 := PressurePoints2 + 1;
				IF PressurePoints2 <= 1000 THEN
					N2PressureValues[PressurePoints2] := NozzlePressure2;
				END_IF
			END_IF

			IF Counter > LatchedNozzleEndCycles1 THEN
				OpenValve1 := FALSE;
				OpenValve2 := FALSE;
				OpenValve3 := FALSE;
				OpenValve4 := FALSE;
				OpenValve17 := FALSE;
				OpenValve18 := FALSE;

				IF PressurePoints > 0 THEN
					AvgPressure := PressureSum / TO_REAL(PressurePoints);
					IF PressurePoints1 > 0 THEN
						AvgPressureN1 := PressureSum1 / TO_REAL(PressurePoints1);
					ELSE
						AvgPressureN1 := 0.0;
					END_IF
					IF PressurePoints2 > 0 THEN
						AvgPressureN2 := PressureSum2 / TO_REAL(PressurePoints2);
					ELSE
						AvgPressureN2 := 0.0;
					END_IF
					ShotCounter := ShotCounter + 1;
					LogPressureTrigger := TRUE;
				END_IF
				IF GuiReorientationControlActive AND (BatchActiveSequence[1] > 0) THEN
					BatchSlotIndex := UDINT_TO_INT((BatchActiveSequence[1] - 1) MOD 128);
					BatchQueueFinishedMask[BatchSlotIndex] := BatchQueueFinishedMask[BatchSlotIndex] OR BYTE#1;
					BatchActiveSequence[1] := 0;
					GuiArrayEnabled1 := FALSE;
				END_IF

				Counter := 0;
				State := 2;
			END_IF
		END_IF
		
	6:
		Enable0 := FALSE;
		Acknowledge0 := FALSE;
		OpenValve1 := FALSE;
		OpenValve2 := FALSE;
		OpenValve3 := FALSE;
		OpenValve4 := FALSE;
		OpenValve17 := FALSE;
		OpenValve18 := FALSE;
END_CASE

CASE State2 OF
	2:
		//start nozzle array 2 on the falling edge of light barrier 4
		IF NOT Array2Active THEN
			Array2TriggerPending := FALSE;
		ELSIF Array2TriggerPending THEN
			Array2TriggerPending := FALSE;
			Counter2 := 0;
			LatchedDelayCycles2 := DelayDurationCycles2;
			LatchedNozzleEndCycles2 := DelayDurationCycles2 + ShotDurationCycles2;
			State2 := State2 + 1;
		END_IF
	3:
		IF NOT Array2Active THEN
			OpenValve5 := FALSE;
			OpenValve6 := FALSE;
			OpenValve7 := FALSE;
			OpenValve8 := FALSE;
			OpenValve19 := FALSE;
			OpenValve20 := FALSE;
			Counter2 := 0;
			State2 := 2;
		ELSE
			Counter2 := Counter2 + 1;
			OpenValve5 := GuiArrayEnabled2 AND GuiNozzleEnabled7 AND (Counter2 > LatchedDelayCycles2) AND (Counter2 <= LatchedNozzleEndCycles2);
			OpenValve6 := GuiArrayEnabled2 AND GuiNozzleEnabled8 AND (Counter2 > LatchedDelayCycles2) AND (Counter2 <= LatchedNozzleEndCycles2);
			OpenValve7 := GuiArrayEnabled2 AND GuiNozzleEnabled9 AND (Counter2 > LatchedDelayCycles2) AND (Counter2 <= LatchedNozzleEndCycles2);
			OpenValve8 := GuiArrayEnabled2 AND GuiNozzleEnabled10 AND (Counter2 > LatchedDelayCycles2) AND (Counter2 <= LatchedNozzleEndCycles2);
			OpenValve19 := GuiArrayEnabled2 AND GuiNozzleEnabled11 AND (Counter2 > LatchedDelayCycles2) AND (Counter2 <= LatchedNozzleEndCycles2);
			OpenValve20 := GuiArrayEnabled2 AND GuiNozzleEnabled12 AND (Counter2 > LatchedDelayCycles2) AND (Counter2 <= LatchedNozzleEndCycles2);
			IF GuiReorientationControlActive AND (BatchActiveSequence[2] > 0)
				AND (OpenValve5 OR OpenValve6 OR OpenValve7 OR OpenValve8 OR OpenValve19 OR OpenValve20) THEN
				BatchSlotIndex := UDINT_TO_INT((BatchActiveSequence[2] - 1) MOD 128);
				BatchQueueActuatedMask[BatchSlotIndex] := BatchQueueActuatedMask[BatchSlotIndex] OR BYTE#2;
			END_IF

			IF Counter2 > LatchedNozzleEndCycles2 THEN
				OpenValve5 := FALSE;
				OpenValve6 := FALSE;
				OpenValve7 := FALSE;
				OpenValve8 := FALSE;
				OpenValve19 := FALSE;
				OpenValve20 := FALSE;
				IF GuiReorientationControlActive AND (BatchActiveSequence[2] > 0) THEN
					BatchSlotIndex := UDINT_TO_INT((BatchActiveSequence[2] - 1) MOD 128);
					BatchQueueFinishedMask[BatchSlotIndex] := BatchQueueFinishedMask[BatchSlotIndex] OR BYTE#2;
					BatchActiveSequence[2] := 0;
					GuiArrayEnabled2 := FALSE;
				END_IF
				Counter2 := 0;
				State2 := 2;
			END_IF
		END_IF
END_CASE

CASE State3 OF
	0:
		Enable1 := TRUE;
		Acknowledge1 := FALSE;
		State3 := State3 + 1;

	1:
		Enable1 := TRUE;
		Acknowledge1 := TRUE;
		State3 := State3 + 1;

	2:
		//start nozzle array 3 on the falling edge of light barrier 6
		IF NOT Array3Active THEN
			Array3TriggerPending := FALSE;
		ELSIF Array3TriggerPending THEN
			Array3TriggerPending := FALSE;
			Counter3 := 0;
			LatchedDelayCycles3 := DelayDurationCycles3;
			LatchedNozzleEndCycles3 := DelayDurationCycles3 + ShotDurationCycles3;
			State3 := State3 + 1;
		END_IF

	3:
		IF NOT Array3Active THEN
			OpenValve9 := FALSE;
			OpenValve10 := FALSE;
			OpenValve11 := FALSE;
			OpenValve12 := FALSE;
			OpenValve21 := FALSE;
			OpenValve22 := FALSE;
			Counter3 := 0;
			State3 := 2;
		ELSE
			Counter3 := Counter3 + 1;
			OpenValve9 := GuiArrayEnabled3 AND GuiNozzleEnabled13 AND (Counter3 > LatchedDelayCycles3) AND (Counter3 <= LatchedNozzleEndCycles3);
			OpenValve10 := GuiArrayEnabled3 AND GuiNozzleEnabled14 AND (Counter3 > LatchedDelayCycles3) AND (Counter3 <= LatchedNozzleEndCycles3);
			OpenValve11 := GuiArrayEnabled3 AND GuiNozzleEnabled15 AND (Counter3 > LatchedDelayCycles3) AND (Counter3 <= LatchedNozzleEndCycles3);
			OpenValve12 := GuiArrayEnabled3 AND GuiNozzleEnabled16 AND (Counter3 > LatchedDelayCycles3) AND (Counter3 <= LatchedNozzleEndCycles3);
			OpenValve21 := GuiArrayEnabled3 AND GuiNozzleEnabled17 AND (Counter3 > LatchedDelayCycles3) AND (Counter3 <= LatchedNozzleEndCycles3);
			OpenValve22 := GuiArrayEnabled3 AND GuiNozzleEnabled18 AND (Counter3 > LatchedDelayCycles3) AND (Counter3 <= LatchedNozzleEndCycles3);
			IF GuiReorientationControlActive AND (BatchActiveSequence[3] > 0)
				AND (OpenValve9 OR OpenValve10 OR OpenValve11 OR OpenValve12 OR OpenValve21 OR OpenValve22) THEN
				BatchSlotIndex := UDINT_TO_INT((BatchActiveSequence[3] - 1) MOD 128);
				BatchQueueActuatedMask[BatchSlotIndex] := BatchQueueActuatedMask[BatchSlotIndex] OR BYTE#4;
			END_IF

			IF Counter3 > LatchedNozzleEndCycles3 THEN
				OpenValve9 := FALSE;
				OpenValve10 := FALSE;
				OpenValve11 := FALSE;
				OpenValve12 := FALSE;
				OpenValve21 := FALSE;
				OpenValve22 := FALSE;
				IF GuiReorientationControlActive AND (BatchActiveSequence[3] > 0) THEN
					BatchSlotIndex := UDINT_TO_INT((BatchActiveSequence[3] - 1) MOD 128);
					BatchQueueFinishedMask[BatchSlotIndex] := BatchQueueFinishedMask[BatchSlotIndex] OR BYTE#4;
					BatchActiveSequence[3] := 0;
					GuiArrayEnabled3 := FALSE;
				END_IF
				Counter3 := 0;
				State3 := 2;
			END_IF
		END_IF

	6:
		Enable1 := FALSE;
		Acknowledge1 := FALSE;
		OpenValve9 := FALSE;
		OpenValve10 := FALSE;
		OpenValve11 := FALSE;
		OpenValve12 := FALSE;
		OpenValve21 := FALSE;
		OpenValve22 := FALSE;
END_CASE

CASE State4 OF
	2:
		//start nozzle array 4 on the falling edge of light barrier 8
		IF NOT Array4Active THEN
			Array4TriggerPending := FALSE;
		ELSIF Array4TriggerPending THEN
			Array4TriggerPending := FALSE;
			Counter4 := 0;
			LatchedDelayCycles4 := DelayDurationCycles4;
			LatchedNozzleEndCycles4 := DelayDurationCycles4 + ShotDurationCycles4;
			State4 := State4 + 1;
		END_IF

	3:
		IF NOT Array4Active THEN
			OpenValve13 := FALSE;
			OpenValve14 := FALSE;
			OpenValve15 := FALSE;
			OpenValve16 := FALSE;
			OpenValve23 := FALSE;
			OpenValve24 := FALSE;
			Counter4 := 0;
			State4 := 2;
		ELSE
			Counter4 := Counter4 + 1;
			OpenValve13 := GuiArrayEnabled4 AND GuiNozzleEnabled19 AND (Counter4 > LatchedDelayCycles4) AND (Counter4 <= LatchedNozzleEndCycles4);
			OpenValve14 := GuiArrayEnabled4 AND GuiNozzleEnabled20 AND (Counter4 > LatchedDelayCycles4) AND (Counter4 <= LatchedNozzleEndCycles4);
			OpenValve15 := GuiArrayEnabled4 AND GuiNozzleEnabled21 AND (Counter4 > LatchedDelayCycles4) AND (Counter4 <= LatchedNozzleEndCycles4);
			OpenValve16 := GuiArrayEnabled4 AND GuiNozzleEnabled22 AND (Counter4 > LatchedDelayCycles4) AND (Counter4 <= LatchedNozzleEndCycles4);
			OpenValve23 := GuiArrayEnabled4 AND GuiNozzleEnabled23 AND (Counter4 > LatchedDelayCycles4) AND (Counter4 <= LatchedNozzleEndCycles4);
			OpenValve24 := GuiArrayEnabled4 AND GuiNozzleEnabled24 AND (Counter4 > LatchedDelayCycles4) AND (Counter4 <= LatchedNozzleEndCycles4);
			IF GuiReorientationControlActive AND (BatchActiveSequence[4] > 0)
				AND (OpenValve13 OR OpenValve14 OR OpenValve15 OR OpenValve16 OR OpenValve23 OR OpenValve24) THEN
				BatchSlotIndex := UDINT_TO_INT((BatchActiveSequence[4] - 1) MOD 128);
				BatchQueueActuatedMask[BatchSlotIndex] := BatchQueueActuatedMask[BatchSlotIndex] OR BYTE#8;
			END_IF

			IF Counter4 > LatchedNozzleEndCycles4 THEN
				OpenValve13 := FALSE;
				OpenValve14 := FALSE;
				OpenValve15 := FALSE;
				OpenValve16 := FALSE;
				OpenValve23 := FALSE;
				OpenValve24 := FALSE;
				IF GuiReorientationControlActive AND (BatchActiveSequence[4] > 0) THEN
					BatchSlotIndex := UDINT_TO_INT((BatchActiveSequence[4] - 1) MOD 128);
					BatchQueueFinishedMask[BatchSlotIndex] := BatchQueueFinishedMask[BatchSlotIndex] OR BYTE#8;
					BatchActiveSequence[4] := 0;
					GuiArrayEnabled4 := FALSE;
				END_IF
				Counter4 := 0;
				State4 := 2;
			END_IF
		END_IF
END_CASE

// Physical idle status covers the four active jobs and all queued array jobs.
ReorientationArraysIdle := (State = 2) AND (State2 = 2) AND (State3 = 2) AND (State4 = 2)
	AND NOT Array1TriggerPending AND NOT Array2TriggerPending AND NOT Array3TriggerPending AND NOT Array4TriggerPending
	AND (BatchJobCount[1] = 0) AND (BatchJobCount[2] = 0) AND (BatchJobCount[3] = 0) AND (BatchJobCount[4] = 0)
	AND (BatchActiveSequence[1] = 0) AND (BatchActiveSequence[2] = 0)
	AND (BatchActiveSequence[3] = 0) AND (BatchActiveSequence[4] = 0)
	AND NOT OpenValve1 AND NOT OpenValve2 AND NOT OpenValve3 AND NOT OpenValve4
	AND NOT OpenValve5 AND NOT OpenValve6 AND NOT OpenValve7 AND NOT OpenValve8
	AND NOT OpenValve9 AND NOT OpenValve10 AND NOT OpenValve11 AND NOT OpenValve12
	AND NOT OpenValve13 AND NOT OpenValve14 AND NOT OpenValve15 AND NOT OpenValve16
	AND NOT OpenValve17 AND NOT OpenValve18 AND NOT OpenValve19 AND NOT OpenValve20
	AND NOT OpenValve21 AND NOT OpenValve22 AND NOT OpenValve23 AND NOT OpenValve24;
// Complete records strictly in sequence.  LB8 may arrive before a delayed array
// pulse ends, therefore ExitSeen and all four finished bits are both required.
IF GuiReorientationControlActive AND ((ReorientationState = 20) OR (ReorientationState = 30))
	AND (BatchNextCompleteSequence <= ReorientationQueueEnqueueAck) THEN
	BatchSlotIndex := UDINT_TO_INT((BatchNextCompleteSequence - 1) MOD 128);
	IF BatchQueueExitSeen[BatchSlotIndex] AND (BatchQueueFinishedMask[BatchSlotIndex] = BYTE#15) THEN
		BatchResultSequence[BatchSlotIndex] := BatchQueueSequence[BatchSlotIndex];
		BatchResultTriggeredMask[BatchSlotIndex] := BatchQueueTriggeredMask[BatchSlotIndex];
		BatchResultFaultCode[BatchSlotIndex] := 0;
		ReorientationQueueCompletedCount := BatchNextCompleteSequence;
		ReorientationCycleCounter := ReorientationCycleCounter + 1;
		IF BatchQueueArrayMask[BatchSlotIndex] = BYTE#0 THEN
			ReorientationQueueBypassCount := ReorientationQueueBypassCount + 1;
		END_IF
		BatchNextCompleteSequence := BatchNextCompleteSequence + 1;
	END_IF
END_IF

// Result ring head. The GUI acknowledges only after its image/CSV export.
IF BatchAcceptedResultAck < ReorientationQueueCompletedCount THEN
	BatchSlotIndex := UDINT_TO_INT(BatchAcceptedResultAck MOD 128);
	ReorientationResultAvailable := TRUE;
	ReorientationResultSequence := BatchResultSequence[BatchSlotIndex];
	ReorientationResultTriggeredMask := BatchResultTriggeredMask[BatchSlotIndex];
	ReorientationResultFaultCode := BatchResultFaultCode[BatchSlotIndex];
ELSE
	ReorientationResultAvailable := FALSE;
END_IF

// A normal finish drains sensors, array FIFOs and exported results before the
// conveyor is stopped. No timeout is imposed on an intentionally long run.
IF GuiReorientationControlActive AND (ReorientationState = 30)
	AND (ReorientationQueueCompletedCount = ReorientationQueueEnqueueAck)
	AND (BatchAcceptedResultAck = ReorientationQueueCompletedCount)
	AND ReorientationArraysIdle THEN
	GuiConveyorEnabled := FALSE;
	ReorientationComplete := TRUE;
	ReorientationState := 40;
END_IF

ReorientationBusy := GuiReorientationControlActive AND (ReorientationState >= 10) AND (ReorientationState < 40);

// Hard close on abort/watchdog/timeout; retained profile values are harmless while
// the enables and conveyor permit remain latched off.
IF ReorientationSafeLatch THEN
	Counter := 0; Counter2 := 0; Counter3 := 0; Counter4 := 0;
	BatchJobCount[1] := 0; BatchJobCount[2] := 0; BatchJobCount[3] := 0; BatchJobCount[4] := 0;
	BatchActiveSequence[1] := 0; BatchActiveSequence[2] := 0;
	BatchActiveSequence[3] := 0; BatchActiveSequence[4] := 0;
	IF State = 3 THEN State := 2; END_IF
	IF State2 = 3 THEN State2 := 2; END_IF
	IF State3 = 3 THEN State3 := 2; END_IF
	IF State4 = 3 THEN State4 := 2; END_IF
	OpenValve1 := FALSE; OpenValve2 := FALSE; OpenValve3 := FALSE; OpenValve4 := FALSE;
	OpenValve5 := FALSE; OpenValve6 := FALSE; OpenValve7 := FALSE; OpenValve8 := FALSE;
	OpenValve9 := FALSE; OpenValve10 := FALSE; OpenValve11 := FALSE; OpenValve12 := FALSE;
	OpenValve13 := FALSE; OpenValve14 := FALSE; OpenValve15 := FALSE; OpenValve16 := FALSE;
	OpenValve17 := FALSE; OpenValve18 := FALSE; OpenValve19 := FALSE; OpenValve20 := FALSE;
	OpenValve21 := FALSE; OpenValve22 := FALSE; OpenValve23 := FALSE; OpenValve24 := FALSE;
END_IF

// Setup movement must never trigger a nozzle, even if a state was active on entry.
IF GuiConveyorCalibrationMode OR GuiVelocityCheckMode THEN
	Array1TriggerPending := FALSE;
	Array2TriggerPending := FALSE;
	Array3TriggerPending := FALSE;
	Array4TriggerPending := FALSE;
	Counter := 0;
	Counter2 := 0;
	Counter3 := 0;
	Counter4 := 0;
	IF State = 3 THEN State := 2; END_IF
	IF State2 = 3 THEN State2 := 2; END_IF
	IF State3 = 3 THEN State3 := 2; END_IF
	IF State4 = 3 THEN State4 := 2; END_IF
	OpenValve1 := FALSE;
	OpenValve2 := FALSE;
	OpenValve3 := FALSE;
	OpenValve4 := FALSE;
	OpenValve5 := FALSE;
	OpenValve6 := FALSE;
	OpenValve7 := FALSE;
	OpenValve8 := FALSE;
	OpenValve9 := FALSE;
	OpenValve10 := FALSE;
	OpenValve11 := FALSE;
	OpenValve12 := FALSE;
	OpenValve13 := FALSE;
	OpenValve14 := FALSE;
	OpenValve15 := FALSE;
	OpenValve16 := FALSE;
	OpenValve17 := FALSE;
	OpenValve18 := FALSE;
	OpenValve19 := FALSE;
	OpenValve20 := FALSE;
	OpenValve21 := FALSE;
	OpenValve22 := FALSE;
	OpenValve23 := FALSE;
	OpenValve24 := FALSE;
END_IF

FBValveControlV0(
	awBusDataFromVTEM:= Valve0_IN, 
	awBusDataToVTEM:= Valve0_OUT, 
	xEnable:= Enable0, 
	bySetValveMode:= ValveMode0, 
	bySetAppControl:= AppControl0, 
	bySetAppOption:= AppOption0, 
	iSetpointValue1:= PresValueV02, 
	iSetpointValue2:= PresValueV04, 
	xManualAcknowledge:= Acknowledge0, 
	byActualValveMode=> ActValveMode0, 
	byActualValveState=> ActValveState0, 
	byActualAppState=> ActAppState0, 
	iActualValue1=> ActPresValueV02, 
	iActualValue2=> ActPresValueV04, 
	iResponseToValveModeSet=> ResponseToValveModeSet0, 
	iErrorCode=> ErrorCode0);

FBValveControlV1(
	awBusDataFromVTEM:= Valve1_IN,
	awBusDataToVTEM:= Valve1_OUT,
	xEnable:= Enable1,
	bySetValveMode:= ValveMode1,
	bySetAppControl:= AppControl1,
	bySetAppOption:= AppOption1,
	iSetpointValue1:= PresValueV12,
	iSetpointValue2:= PresValueV14,
	xManualAcknowledge:= Acknowledge1,
	byActualValveMode=> ActValveMode1,
	byActualValveState=> ActValveState1,
	byActualAppState=> ActAppState1,
	iActualValue1=> ActPresValueV12,
	iActualValue2=> ActPresValueV14,
	iResponseToValveModeSet=> ResponseToValveModeSet1,
	iErrorCode=> ErrorCode1);

LastLightBarrier1 := LightBarrierStable1;
LastLightBarrier2 := LightBarrierStable2;
LastLightBarrier3 := LightBarrierStable3;
LastLightBarrier4 := LightBarrierStable4;
LastLightBarrier5 := LightBarrierStable5;
LastLightBarrier6 := LightBarrierStable6;
LastLightBarrier7 := LightBarrierStable7;
LastLightBarrier8 := LightBarrierStable8;

// Call once, last in the 1 ms cycle, so late batch completion/abort also reaches both drives.
IF (ConveyorMotionMode = 1) AND NOT GuiConveyorEnabled THEN
	StepperPosExecute := FALSE;
END_IF
IF ConveyorServoStopRequested THEN
	GuiConveyorEnabled := FALSE;
END_IF
// The old positioning-interface "emergency stop" flag is also used by ordinary
// GUI Stop/calibration exit. Request a controlled ramp and wait for measured standstill.
IF StepperPosEmergencyStop OR ConveyorServoStopRequested THEN
	StepperPosExecute := FALSE;
END_IF
IF ReorientationSafeLatch OR NOT ConveyorServoCommissioned THEN
	StepperControlEnable := FALSE;
	StepperPosExecute := FALSE;
END_IF
// A reset always cancels outstanding commands. It cannot restart either motor.
IF ConveyorServoResetRequested THEN
	GuiConveyorEnabled := FALSE;
	GuiConveyorCalibrationMode := FALSE;
	StepperControlEnable := FALSE;
	StepperPosExecute := FALSE;
	StepperPosEmergencyStop := FALSE;
	ConveyorMotionState := 0;
	ConveyorMotionMode := 0;
	CalibrationBusy := FALSE;
	CalibrationLeftMarkValid := FALSE;
	CalibrationRightMarkValid := FALSE;
END_IF

TandemConveyor(
	MotorCount := 1, // Device 3 has one physical servo; unused motor 2 stays disabled.
	Enable := StepperControlEnable,
	Execute := StepperPosExecute,
	EmergencyStop := FALSE, // application cancellation ramps through Execute; faults override in FB
	Reset := ConveyorServoResetRequested,
	Inhibit := ReorientationSafeLatch,
	StartType := StepperPosStartType,
	TargetPosition := StepperPosTargetPosition,
	Velocity := StepperPosVelocity,
	LegacySpeedRange := REAL_TO_LREAL(ConveyorSpeedRangeFullStepsPerSec),
	Commissioned := ConveyorServoCommissioned AND ConveyorDriveSettings.Valid,
	Direction1 := ConveyorServoDirection1,
	Direction2 := ConveyorServoDirection2,
	Motor2Ratio := ConveyorServoMotor2Ratio,
	FeedbackCountsPerRev := ConveyorServoFeedbackCountsPerRev,
	FeedbackCountsPerRev2 := ConveyorServoFeedbackCountsPerRev2,
	VelocityUnitsPerRevPerSec := ConveyorServoVelocityUnitsPerRevPerSec,
	VelocityUnitsPerRevPerSec2 := ConveyorServoVelocityUnitsPerRevPerSec2,
	MaxMotorRpm := ConveyorServoMaxMotorRpm,
	AccelerationRpmPerSec := ConveyorServoAccelerationRpmPerSec,
	PositionGain := ConveyorServoPositionGain,
	SyncToleranceFullSteps := ConveyorServoSyncToleranceFullSteps,
	FollowingToleranceFullSteps := ConveyorServoFollowingToleranceFullSteps,
	CycleSeconds := 0.001,
	Position1 := ConveyorServo1Position,
	Position2 := ConveyorServo2Position,
	Statusword1 := ConveyorServo1Statusword,
	Statusword2 := ConveyorServo2Statusword,
	WcState1 := ConveyorServo1WcState,
	WcState2 := ConveyorServo2WcState,
	InfoState1 := ConveyorServo1InfoState,
	InfoState2 := ConveyorServo2InfoState,
	ActualVelocity1 := ConveyorServo1ActualVelocity,
	ActualVelocity2 := ConveyorServo2ActualVelocity,
	FeedbackInvalid1 := ConveyorServo1FeedbackInvalid,
	FeedbackInvalid2 := ConveyorServo2FeedbackInvalid,
	Controlword1 => ConveyorServo1Controlword,
	Controlword2 => ConveyorServo2Controlword,
	TargetVelocity1 => ConveyorServo1TargetVelocity,
	TargetVelocity2 => ConveyorServo2TargetVelocity,
	LegacyPosition => StepperInternalPosition,
	Busy => StepperPosBusy,
	InTarget => StepperPosInTarget,
	Ready => StepperPosReadyToExecute,
	Warning => StepperPosWarning,
	Error => StepperPosError,
	FaultCode => ConveyorServoFaultCode,
	StmStatus => StepperStmStatus,
	State => ConveyorServoState,
	SyncErrorFullSteps => ConveyorServoSyncErrorFullSteps);
CalibrationError := StepperPosError;
IF StepperPosError THEN
	GuiConveyorEnabled := FALSE;
	GuiConveyorCalibrationMode := FALSE;
	CalibrationStatusCode := 5;
END_IF

END_PROGRAM

// ---- POUs/FB_TandemConveyor.TcPOU
FUNCTION_BLOCK FB_TandemConveyor
VAR_INPUT
    MotorCount : UINT := 2; //1 single conveyor; 2 tandem. Frozen at commissioning.
    Enable                  : BOOL;
    Execute                 : BOOL;
    EmergencyStop           : BOOL;
    Reset                   : BOOL;
    Inhibit                 : BOOL;
    StartType               : UINT; //2 signed relative increments; 3 endless+; 4 endless-
    TargetPosition          : UDINT; //signed DINT bit pattern, 64 increments/virtual full step
    Velocity                : INT; //positive 1..10000, fraction of LegacySpeedRange
    LegacySpeedRange         : LREAL := 2000.0; //virtual full steps/s at Velocity=10000

    //Commissioning is independent of the GUI's writable calibration-valid flag.
    //The drive must already be commissioned in CSV mode (MDP742 mode 9).
    Commissioned            : BOOL := FALSE;
    Direction1              : INT := 0; //must be explicitly commissioned as -1 or +1
    Direction2              : INT := 0;
    Motor2Ratio             : LREAL := 1.0; //motor2 revolutions per motor1 revolution
    FeedbackCountsPerRev    : LREAL := 1048576.0; //verify actual configured PDO resolution
    FeedbackCountsPerRev2   : LREAL := 1048576.0;
    VelocityUnitsPerRevPerSec : LREAL := 0.0; //REQUIRED verified CSV raw velocity scaling
    VelocityUnitsPerRevPerSec2 : LREAL := 0.0;
    MaxMotorRpm             : LREAL := 300.0;
    AccelerationRpmPerSec    : LREAL := 300.0;
    PositionGain            : LREAL := 5.0; //1/s, bounded position correction around common trajectory
    SyncToleranceFullSteps  : LREAL := 5.0;
    FollowingToleranceFullSteps : LREAL := 20.0;
    CycleSeconds            : LREAL := 0.001; //must match the calling PLC task

    Position1               : UDINT;
    Position2               : UDINT;
    Statusword1             : UINT;
    Statusword2             : UINT;
    WcState1                : BOOL;
    WcState2                : BOOL;
    InfoState1              : UINT;
    InfoState2              : UINT;
    ActualVelocity1         : DINT; //same raw units as TargetVelocity
    ActualVelocity2         : DINT;
    FeedbackInvalid1        : BOOL; //FB status TxPDO State, when mapped
    FeedbackInvalid2        : BOOL;
END_VAR
VAR_OUTPUT
    Controlword1            : UINT;
    Controlword2            : UINT;
    TargetVelocity1         : DINT;
    TargetVelocity2         : DINT;
    LegacyPosition          : UDINT; //measured motor1, 200 virtual full steps/rev * 64 increments
    Busy                    : BOOL;
    InTarget                : BOOL;
    Ready                   : BOOL;
    Warning                 : BOOL;
    Error                   : BOOL;
    //Latched: 1 invalid configuration, 2 drive fault, 3 EtherCAT/feedback invalid,
    //4 enable timeout, 5 synchronization, 6 following/operation lost,
    //7 move/stop timeout, 8 configuration changed, 9 reset timeout, 10 invalid command.
    FaultCode               : UINT;
    //Compatibility summary only: bit0 ready, bit1 busy, bit3 fault, bit7 warning.
    StmStatus               : WORD;
    //0 disabled, 10 enabling, 20 ready, 30 moving, 40 decelerating, 80 resetting, 90 fault.
    State                   : UINT;
    SyncErrorFullSteps      : LREAL;
END_VAR
VAR
    ActiveCount : INT;
    CfgMotorCount : UINT;
    RawPosition             : ARRAY[1..2] OF UDINT;
    PreviousPosition        : ARRAY[1..2] OF UDINT;
    RawStatus               : ARRAY[1..2] OF UINT;
    RawActualVelocity       : ARRAY[1..2] OF DINT;
    DriveControl            : ARRAY[1..2] OF UINT;
    DriveEnableStep         : ARRAY[1..2] OF UINT;
    MeasuredPosition        : ARRAY[1..2] OF LREAL; //normalized common virtual full steps
    MeasuredVelocity        : ARRAY[1..2] OF LREAL;
    DriveCommand            : ARRAY[1..2] OF LREAL;
    CfgDirection            : ARRAY[1..2] OF INT;
    CfgRatio                : ARRAY[1..2] OF LREAL;
    CfgFeedbackCounts       : ARRAY[1..2] OF LREAL;
    CfgVelocityUnits        : ARRAY[1..2] OF LREAL;
    CfgMaxRpm               : LREAL;
    CfgAccelerationRpm      : LREAL;
    CfgGain                 : LREAL;
    CfgSyncTolerance        : LREAL;
    CfgFollowingTolerance   : LREAL;
    CfgCycle                : LREAL;
    CfgLegacyRange          : LREAL;
    ConfigLoaded            : BOOL;
    ConfigValid             : BOOL;
    ConfigUnchanged         : BOOL;
    CaptureConfig           : BOOL;
    HealthyInputs           : BOOL;
    StartupComplete         : BOOL;
    StandstillInitialized   : BOOL;
    StandstillOrigin        : ARRAY[1..2] OF UDINT;
    StandstillCounts        : ARRAY[1..2] OF LREAL;
    WithinStandstillWindow  : BOOL;
    EncoderStationary       : BOOL;
    DriveFault              : BOOL;
    AllEnabled              : BOOL;
    WantDriveEnable         : BOOL;
    FeedbackInitialized     : BOOL;
    RebaseRequested         : BOOL;
    RestartBlocked          : BOOL := TRUE;
    ResetActive             : BOOL;
    ResetPulse              : BOOL;
    ResetEdge               : BOOL;
    ExecuteEdge             : BOOL;
    LastReset               : BOOL;
    LastExecute             : BOOL;
    PositionSettled         : BOOL;
    SpeedSettled            : BOOL;
    CompletedThisCycle      : BOOL;
    FiniteMove              : BOOL;
    LimitedSpeed            : BOOL;
    FollowingExceeded       : BOOL;
    StopTimerStart           : BOOL;
    I                       : INT;
    MaskedStatus            : UINT;
    EncoderDelta            : LINT;
    SignedTarget            : LINT;
    LegacyIncrements        : LINT;
    WrappedIncrements       : LINT;
    MaxCommonSpeed          : LREAL;
    CommonAcceleration      : LREAL;
    CommandSpeed            : LREAL;
    CommandDirection        : LREAL;
    TrajectoryPosition      : LREAL;
    TrajectoryVelocity      : LREAL;
    TargetFullSteps         : LREAL;
    DesiredVelocity         : LREAL;
    PreviousTrajectoryVelocity : LREAL;
    NextTrajectoryPosition  : LREAL;
    Remaining               : LREAL;
    BrakingSpeed            : LREAL;
    VelocityIncrement       : LREAL;
    PositionError           : LREAL;
    Correction              : LREAL;
    CorrectionLimit         : LREAL;
    RawCommand              : LREAL;
    DurationMs              : LREAL;
    MoveTimeout             : TIME := T#10S;
    StopTimeout             : TIME := T#10S;
    EnableTimer             : TON;
    SyncTimer               : TON;
    FollowingTimer          : TON;
    SettleTimer             : TON;
    MoveTimer               : TON;
    StopTimer               : TON;
    ResetTimer              : TON;
    StartupHealthyTimer     : TON;
    StartupTimeoutTimer     : TON;
    EncoderStandstillTimer  : TON;
END_VAR

//Software coordination/monitoring only. This FB does not implement STO or a safety stop.
//No movement is authorized by default. Configure drive motor/encoder/brake/current,
//CSV mode, PDO mapping, raw scales, gearing/direction and independent machine safety first.
//All configuration is frozen while commissioned; a change requires an idle explicit reset.

Controlword1 := 0;
Controlword2 := 0;
TargetVelocity1 := 0;
TargetVelocity2 := 0;
Ready := FALSE;
Busy := FALSE;
ResetPulse := FALSE;
CaptureConfig := FALSE;
CompletedThisCycle := FALSE;
StopTimerStart := FALSE;
PositionSettled := FALSE;
FollowingExceeded := FALSE;
ResetEdge := Reset AND NOT LastReset;
ExecuteEdge := Execute AND NOT LastExecute;
LastReset := Reset;
LastExecute := Execute;

ActiveCount := 2;
IF ConfigLoaded THEN
    IF CfgMotorCount = 1 THEN ActiveCount := 1; END_IF;
ELSIF MotorCount = 1 THEN ActiveCount := 1; END_IF;
RawPosition[1] := Position1;
RawPosition[2] := Position2;
RawStatus[1] := Statusword1;
RawStatus[2] := Statusword2;
RawActualVelocity[1] := ActualVelocity1;
RawActualVelocity[2] := ActualVelocity2;
FOR I := 1 TO ActiveCount DO
    DriveControl[I] := 0;
    DriveCommand[I] := 0.0;
END_FOR;

//Bounded comparisons also reject NaN and infinity before any conversion or division.
ConfigValid := ((MotorCount = 1) OR (MotorCount = 2))
    AND ((Direction1 = 1) OR (Direction1 = -1))
    AND ((Direction2 = 1) OR (Direction2 = -1))
    AND (Motor2Ratio >= 0.0001) AND (Motor2Ratio <= 10000.0)
    AND (FeedbackCountsPerRev >= 1.0) AND (FeedbackCountsPerRev <= 4294967295.0)
    AND (FeedbackCountsPerRev2 >= 1.0) AND (FeedbackCountsPerRev2 <= 4294967295.0)
    AND (VelocityUnitsPerRevPerSec >= 0.000001) AND (VelocityUnitsPerRevPerSec <= 1000000000.0)
    AND (VelocityUnitsPerRevPerSec2 >= 0.000001) AND (VelocityUnitsPerRevPerSec2 <= 1000000000.0)
    AND (MaxMotorRpm >= 0.1) AND (MaxMotorRpm <= 10000.0)
    AND (AccelerationRpmPerSec >= 0.1) AND (AccelerationRpmPerSec <= 100000.0)
    AND (PositionGain >= 0.01) AND (PositionGain <= 1000.0)
    AND (SyncToleranceFullSteps > 0.0) AND (SyncToleranceFullSteps <= 1000000.0)
    AND (FollowingToleranceFullSteps > 0.0) AND (FollowingToleranceFullSteps <= 1000000.0)
    AND (CycleSeconds >= 0.0001) AND (CycleSeconds <= 0.1)
    AND (LegacySpeedRange >= 0.01) AND (LegacySpeedRange <= 10000000.0);
IF ConfigValid THEN
    ConfigValid := (MaxMotorRpm / 60.0 * VelocityUnitsPerRevPerSec <= 2147480000.0)
        AND (MaxMotorRpm / 60.0 * VelocityUnitsPerRevPerSec2 <= 2147480000.0)
        AND (MaxMotorRpm / AccelerationRpmPerSec <= 3600.0);
END_IF;

HealthyInputs := NOT WcState1 AND (InfoState1 = 8) AND NOT FeedbackInvalid1
    AND ((ActiveCount = 1) OR (NOT WcState2 AND (InfoState2 = 8) AND NOT FeedbackInvalid2));
DriveFault := ((Statusword1 AND UINT#16#0008) <> 0)
    OR ((ActiveCount = 2) AND ((Statusword2 AND UINT#16#0008) <> 0));
Warning := ((Statusword1 AND UINT#16#0080) <> 0)
    OR ((ActiveCount = 2) AND ((Statusword2 AND UINT#16#0080) <> 0));

//Allow initial EtherCAT startup with both output stages disabled. After the first
//100 ms of valid data, any communication loss latches immediately, even while idle.
StartupHealthyTimer(IN := Commissioned AND HealthyInputs, PT := T#100MS);
IF StartupHealthyTimer.Q THEN
    StartupComplete := TRUE;
END_IF;
StartupTimeoutTimer(IN := Commissioned AND NOT StartupComplete, PT := T#5S);
IF StartupTimeoutTimer.Q AND (FaultCode = 0) THEN
    FaultCode := 3;
END_IF;

//The terminal's instantaneous velocity estimate is noisy even with stationary
//encoders. Qualify standstill from BOTH position traces instead: each must stay
//within 0.05 motor full steps (0.09 degrees) of its fixed anchor for 100 ms.
//Anchors do not slide every scan: sustained movement must restart the timer.
WithinStandstillWindow := FALSE;
IF Commissioned AND ConfigValid AND HealthyInputs THEN
    IF NOT StandstillInitialized
        OR (StandstillCounts[1] <> FeedbackCountsPerRev)
        OR (StandstillCounts[2] <> FeedbackCountsPerRev2) THEN
        StandstillCounts[1] := FeedbackCountsPerRev;
        StandstillCounts[2] := FeedbackCountsPerRev2;
        StandstillInitialized := TRUE;
    ELSE
        WithinStandstillWindow := TRUE;
        FOR I := 1 TO ActiveCount DO
            EncoderDelta := UDINT_TO_LINT(RawPosition[I]) - UDINT_TO_LINT(StandstillOrigin[I]);
            IF EncoderDelta > LINT#2147483647 THEN
                EncoderDelta := EncoderDelta - LINT#4294967296;
            ELSIF EncoderDelta < LINT#-2147483648 THEN
                EncoderDelta := EncoderDelta + LINT#4294967296;
            END_IF;
            IF ABS(LINT_TO_LREAL(EncoderDelta)) > StandstillCounts[I] * 0.05 / 200.0 THEN
                WithinStandstillWindow := FALSE;
            END_IF;
        END_FOR;
    END_IF;
    IF NOT WithinStandstillWindow THEN
        FOR I := 1 TO ActiveCount DO
            StandstillOrigin[I] := RawPosition[I];
        END_FOR;
    END_IF;
ELSE
    StandstillInitialized := FALSE;
END_IF;
EncoderStandstillTimer(IN := WithinStandstillWindow, PT := T#100MS);
EncoderStationary := EncoderStandstillTimer.Q;

ConfigUnchanged := ConfigLoaded AND (MotorCount = CfgMotorCount)
    AND (Direction1 = CfgDirection[1]) AND (Direction2 = CfgDirection[2])
    AND (Motor2Ratio = CfgRatio[2]) AND (FeedbackCountsPerRev = CfgFeedbackCounts[1])
    AND (FeedbackCountsPerRev2 = CfgFeedbackCounts[2])
    AND (VelocityUnitsPerRevPerSec = CfgVelocityUnits[1])
    AND (VelocityUnitsPerRevPerSec2 = CfgVelocityUnits[2])
    AND (MaxMotorRpm = CfgMaxRpm) AND (AccelerationRpmPerSec = CfgAccelerationRpm)
    AND (PositionGain = CfgGain) AND (SyncToleranceFullSteps = CfgSyncTolerance)
    AND (FollowingToleranceFullSteps = CfgFollowingTolerance)
    AND (CycleSeconds = CfgCycle) AND (LegacySpeedRange = CfgLegacyRange);

IF Commissioned THEN
    IF NOT ConfigValid AND (FaultCode = 0) THEN
        FaultCode := 1;
    ELSIF ConfigLoaded AND NOT ConfigUnchanged AND (FaultCode = 0) THEN
        FaultCode := 8;
    END_IF;
    //A stale GUI enable at first commissioning must be diagnosed, not leave the
    //caller waiting indefinitely for Ready. Reset cancels it before configuration capture.
    IF NOT ConfigLoaded AND (Enable OR Execute) AND NOT ResetEdge AND (FaultCode = 0) THEN
        FaultCode := 1;
    END_IF;
END_IF;

//The first configuration may be adopted only with both commands off and stopped feedback.
//Reset may adopt a new configuration, but never while either drive is moving.
IF Commissioned AND ConfigValid AND HealthyInputs AND StartupComplete AND NOT Enable AND NOT Execute
    AND NOT Inhibit AND NOT EmergencyStop THEN
    IF EncoderStationary THEN
        IF ResetEdge THEN
            CaptureConfig := TRUE;
            ResetPulse := TRUE;
            ResetActive := TRUE;
            RestartBlocked := TRUE;
            FeedbackInitialized := FALSE;
            RebaseRequested := FALSE;
            State := 80;
            InTarget := FALSE;
        ELSIF NOT ConfigLoaded AND (FaultCode = 0) AND NOT DriveFault THEN
            CaptureConfig := TRUE;
            RebaseRequested := TRUE;
        END_IF;
    END_IF;
END_IF;

IF CaptureConfig THEN
    CfgMotorCount := MotorCount;
    CfgDirection[1] := Direction1;
    CfgDirection[2] := Direction2;
    CfgRatio[1] := 1.0;
    CfgRatio[2] := Motor2Ratio;
    CfgFeedbackCounts[1] := FeedbackCountsPerRev;
    CfgFeedbackCounts[2] := FeedbackCountsPerRev2;
    CfgVelocityUnits[1] := VelocityUnitsPerRevPerSec;
    CfgVelocityUnits[2] := VelocityUnitsPerRevPerSec2;
    CfgMaxRpm := MaxMotorRpm;
    CfgAccelerationRpm := AccelerationRpmPerSec;
    CfgGain := PositionGain;
    CfgSyncTolerance := SyncToleranceFullSteps;
    CfgFollowingTolerance := FollowingToleranceFullSteps;
    CfgCycle := CycleSeconds;
    CfgLegacyRange := LegacySpeedRange;
    ConfigLoaded := TRUE;
    ConfigUnchanged := TRUE;
    TrajectoryVelocity := 0.0;
    FOR I := 1 TO ActiveCount DO
        DriveEnableStep[I] := 0;
    END_FOR;
END_IF;

SpeedSettled := FALSE;
IF ConfigLoaded THEN
    MaxCommonSpeed := CfgMaxRpm / 60.0 * 200.0;
    CommonAcceleration := CfgAccelerationRpm / 60.0 * 200.0;
    IF (ActiveCount = 2) AND (CfgRatio[2] > 1.0) THEN
        MaxCommonSpeed := MaxCommonSpeed / CfgRatio[2];
        CommonAcceleration := CommonAcceleration / CfgRatio[2];
    END_IF;
    FOR I := 1 TO ActiveCount DO
        MeasuredVelocity[I] := DINT_TO_LREAL(RawActualVelocity[I]) / CfgVelocityUnits[I]
            * 200.0 * INT_TO_LREAL(CfgDirection[I]) / CfgRatio[I];
    END_FOR;
    SpeedSettled := EncoderStationary;
END_IF;

//Invalid cyclic data is latched and invalidates the origin. Recovery cannot silently
//join new encoder values onto old samples. A stopped explicit reset must rebase it.
IF Commissioned AND NOT HealthyInputs THEN
    IF StartupComplete AND (FaultCode = 0) THEN
        FaultCode := 3;
    END_IF;
    FeedbackInitialized := FALSE;
    RebaseRequested := FALSE;
    ResetActive := FALSE;
END_IF;
IF Commissioned AND HealthyInputs AND DriveFault AND NOT ResetActive AND (FaultCode = 0) THEN
    FaultCode := 2;
END_IF;

ResetTimer(IN := ResetActive AND NOT ResetPulse, PT := T#3S);
IF ResetActive AND NOT ResetPulse THEN
    IF NOT Commissioned OR Inhibit OR EmergencyStop OR Enable OR Execute
        OR NOT HealthyInputs OR NOT ConfigUnchanged THEN
        ResetActive := FALSE;
        IF FaultCode = 0 THEN
            FaultCode := 9;
        END_IF;
    ELSIF NOT DriveFault AND SpeedSettled THEN
        ResetActive := FALSE;
        FaultCode := 0;
        RebaseRequested := TRUE;
        State := 0;
    ELSIF ResetTimer.Q THEN
        ResetActive := FALSE;
        FaultCode := 9;
    END_IF;
END_IF;

//Rebase preserves the last published legacy position; movement during invalid data is
//intentionally not inferred. The two actual motor positions establish a fresh common origin.
IF RebaseRequested AND HealthyInputs AND SpeedSettled AND NOT Enable AND NOT Execute
    AND Commissioned AND NOT ResetActive AND (FaultCode = 0) THEN
    FOR I := 1 TO ActiveCount DO
        PreviousPosition[I] := RawPosition[I];
    END_FOR;
    MeasuredPosition[2] := MeasuredPosition[1];
    TrajectoryPosition := MeasuredPosition[1];
    TrajectoryVelocity := 0.0;
    FeedbackInitialized := TRUE;
    RebaseRequested := FALSE;
END_IF;

IF FeedbackInitialized AND HealthyInputs AND ConfigLoaded THEN
    FOR I := 1 TO ActiveCount DO
        //Explicit signed modular subtraction handles both UDINT wrap directions.
        EncoderDelta := UDINT_TO_LINT(RawPosition[I]) - UDINT_TO_LINT(PreviousPosition[I]);
        IF EncoderDelta > LINT#2147483647 THEN
            EncoderDelta := EncoderDelta - LINT#4294967296;
        ELSIF EncoderDelta < LINT#-2147483648 THEN
            EncoderDelta := EncoderDelta + LINT#4294967296;
        END_IF;
        PreviousPosition[I] := RawPosition[I];
        MeasuredPosition[I] := MeasuredPosition[I] + LINT_TO_LREAL(EncoderDelta)
            / CfgFeedbackCounts[I] * 200.0 * INT_TO_LREAL(CfgDirection[I]) / CfgRatio[I];
    END_FOR;
    //The bound protects the subsequent real/integer conversion on very long uptime.
    IF (ABS(MeasuredPosition[1]) <= 1000000000000.0)
        AND (ABS(MeasuredPosition[2]) <= 1000000000000.0) THEN
        LegacyIncrements := LREAL_TO_LINT(MeasuredPosition[1] * 64.0);
        WrappedIncrements := LegacyIncrements MOD LINT#4294967296;
        IF WrappedIncrements < 0 THEN
            WrappedIncrements := WrappedIncrements + LINT#4294967296;
        END_IF;
        LegacyPosition := LINT_TO_UDINT(WrappedIncrements);
    ELSIF FaultCode = 0 THEN
        FaultCode := 6;
    END_IF;
END_IF;
SyncErrorFullSteps := 0.0;
IF ActiveCount = 2 THEN
    SyncErrorFullSteps := MeasuredPosition[1] - MeasuredPosition[2];
END_IF;

//Any hard software inhibit demands an off-command interval before another enable.
IF NOT Commissioned OR Inhibit OR EmergencyStop THEN
    IF Enable OR Execute THEN
        RestartBlocked := TRUE;
    END_IF;
    InTarget := FALSE;
    TrajectoryVelocity := 0.0;
    IF NOT ResetActive THEN
        State := 0;
    END_IF;
END_IF;
//An off interval may be observed while an inhibit is still asserted. Outputs remain
//disabled by the independent inhibit, but the next deliberate command can re-enable.
IF NOT Enable AND NOT Execute AND NOT ResetActive AND (FaultCode = 0) THEN
    RestartBlocked := FALSE;
END_IF;

AllEnabled := FALSE;
WantDriveEnable := FALSE;
IF ConfigLoaded AND FeedbackInitialized AND HealthyInputs AND Commissioned
    AND ConfigUnchanged AND NOT Inhibit AND NOT EmergencyStop AND NOT RestartBlocked
    AND NOT ResetActive AND (FaultCode = 0) THEN

    //An ordinary Execute/Enable fall uses the configured deceleration. The calling
    //PLC may leave Enable on during this phase; both drives remain enabled until settled.
    IF (State = 30) AND (NOT Execute OR NOT Enable) THEN
        State := 40;
        InTarget := FALSE;
        StopTimerStart := TRUE;
        DurationMs := (ABS(TrajectoryVelocity) / CommonAcceleration + 5.0) * 1000.0;
        StopTimeout := UDINT_TO_TIME(LREAL_TO_UDINT(DurationMs));
    END_IF;
    WantDriveEnable := Enable OR (State = 40);
    IF WantDriveEnable THEN
        IF State = 0 THEN
            State := 10;
        END_IF;
        FOR I := 1 TO ActiveCount DO
            //MDP742 EL7201: bit5 is reserved in this revision. Do not use a DS402
            //0x006F/0x0027 mask; the relevant state pattern here is 0x004F/0x0007.
            MaskedStatus := RawStatus[I] AND UINT#16#004F;
            CASE DriveEnableStep[I] OF
                0:
                    DriveControl[I] := 0; //one disabled scan before the enable sequence
                    DriveEnableStep[I] := 1;
                1:
                    DriveControl[I] := 6;
                    IF MaskedStatus = 1 THEN
                        DriveEnableStep[I] := 2;
                    END_IF;
                2:
                    DriveControl[I] := 7;
                    IF MaskedStatus = 3 THEN
                        DriveEnableStep[I] := 3;
                    END_IF;
                3:
                    DriveControl[I] := 15;
                    IF MaskedStatus = 7 THEN
                        DriveEnableStep[I] := 4;
                    END_IF;
                4:
                    DriveControl[I] := 15;
            ELSE
                DriveEnableStep[I] := 0;
            END_CASE;
        END_FOR;
        AllEnabled := (DriveEnableStep[1] = 4) AND ((Statusword1 AND UINT#16#004F) = 7)
            AND ((ActiveCount = 1) OR ((DriveEnableStep[2] = 4) AND ((Statusword2 AND UINT#16#004F) = 7)));
        IF AllEnabled AND (State = 10) THEN
            State := 20;
        ELSIF NOT AllEnabled AND ((State = 20) OR (State = 30) OR (State = 40)) THEN
            FaultCode := 6; //stop the partner immediately if one loses operation enabled
        END_IF;
    ELSE
        State := 0;
        FOR I := 1 TO ActiveCount DO
            DriveEnableStep[I] := 0;
        END_FOR;
    END_IF;

    IF ExecuteEdge AND (FaultCode = 0) THEN
        IF (State <> 20) OR NOT AllEnabled OR NOT Enable
            OR (Velocity <= 0) OR (Velocity > 10000)
            OR ((StartType <> 2) AND (StartType <> 3) AND (StartType <> 4)) THEN
            FaultCode := 10;
        ELSE
            CommandSpeed := INT_TO_LREAL(Velocity) / 10000.0 * CfgLegacyRange;
            LimitedSpeed := CommandSpeed > MaxCommonSpeed;
            IF LimitedSpeed THEN
                CommandSpeed := MaxCommonSpeed;
            END_IF;
            TrajectoryPosition := MeasuredPosition[1];
            TrajectoryVelocity := 0.0;
            FiniteMove := StartType = 2;
            CommandDirection := 1.0;
            IF StartType = 4 THEN
                CommandDirection := -1.0;
            END_IF;
            IF FiniteMove THEN
                SignedTarget := UDINT_TO_LINT(TargetPosition);
                IF SignedTarget > LINT#2147483647 THEN
                    SignedTarget := SignedTarget - LINT#4294967296;
                END_IF;
                TargetFullSteps := MeasuredPosition[1] + LINT_TO_LREAL(SignedTarget) / 64.0;
                //Finite travel watchdog includes acceleration, settling, and a margin.
                DurationMs := (ABS(TargetFullSteps - TrajectoryPosition) / CommandSpeed
                    + 2.0 * CommandSpeed / CommonAcceleration + 10.0) * 1000.0;
                IF DurationMs > 2000000000.0 THEN
                    FaultCode := 10;
                ELSE
                    MoveTimeout := UDINT_TO_TIME(LREAL_TO_UDINT(DurationMs));
                END_IF;
            END_IF;
            IF FaultCode = 0 THEN
                State := 30;
                InTarget := FALSE;
            END_IF;
        END_IF;
    END_IF;

    IF AllEnabled AND (FaultCode = 0) AND ((State = 30) OR (State = 40)) THEN
        DesiredVelocity := 0.0;
        Remaining := TargetFullSteps - TrajectoryPosition;
        IF State = 30 THEN
            IF FiniteMove THEN
                BrakingSpeed := SQRT(2.0 * CommonAcceleration * ABS(Remaining));
                DesiredVelocity := MIN(CommandSpeed, BrakingSpeed);
                IF Remaining < 0.0 THEN
                    DesiredVelocity := -DesiredVelocity;
                END_IF;
            ELSE
                DesiredVelocity := CommandDirection * CommandSpeed;
            END_IF;
        END_IF;
        VelocityIncrement := CommonAcceleration * CfgCycle;
        PreviousTrajectoryVelocity := TrajectoryVelocity;
        IF TrajectoryVelocity < DesiredVelocity THEN
            TrajectoryVelocity := MIN(TrajectoryVelocity + VelocityIncrement, DesiredVelocity);
        ELSIF TrajectoryVelocity > DesiredVelocity THEN
            TrajectoryVelocity := MAX(TrajectoryVelocity - VelocityIncrement, DesiredVelocity);
        END_IF;
        NextTrajectoryPosition := TrajectoryPosition
            + (PreviousTrajectoryVelocity + TrajectoryVelocity) * 0.5 * CfgCycle;
        IF (State = 30) AND FiniteMove
            AND ((Remaining = 0.0) OR ((TargetFullSteps - NextTrajectoryPosition) * Remaining <= 0.0)) THEN
            TrajectoryPosition := TargetFullSteps;
            TrajectoryVelocity := 0.0;
        ELSE
            TrajectoryPosition := NextTrajectoryPosition;
        END_IF;

        //Both position corrections track the same trajectory. Bounded corrections and
        //the final common speed clamp respect each motor's configured RPM limit.
        CorrectionLimit := MaxCommonSpeed * 0.25;
        FOR I := 1 TO ActiveCount DO
            PositionError := TrajectoryPosition - MeasuredPosition[I];
            IF ABS(PositionError) > CfgFollowingTolerance THEN
                FollowingExceeded := TRUE;
            END_IF;
            Correction := LIMIT(-CorrectionLimit, CfgGain * PositionError, CorrectionLimit);
            DriveCommand[I] := LIMIT(-MaxCommonSpeed, TrajectoryVelocity + Correction, MaxCommonSpeed);
        END_FOR;
        IF ABS(TrajectoryVelocity) <= 0.01 THEN
            PositionSettled := (ABS(TrajectoryPosition - MeasuredPosition[1]) <= 0.25)
                AND ((ActiveCount = 1) OR (ABS(TrajectoryPosition - MeasuredPosition[2]) <= 0.25));
        END_IF;
    END_IF;
END_IF;

EnableTimer(IN := WantDriveEnable AND NOT AllEnabled AND (FaultCode = 0), PT := T#5S);
SyncTimer(IN := ((State = 30) OR (State = 40)) AND (FaultCode = 0)
    AND (ABS(SyncErrorFullSteps) > CfgSyncTolerance), PT := T#250MS);
FollowingTimer(IN := FollowingExceeded AND (FaultCode = 0), PT := T#250MS);
SettleTimer(IN := ((State = 40) OR ((State = 30) AND FiniteMove))
    AND PositionSettled AND SpeedSettled AND (FaultCode = 0), PT := T#100MS);
MoveTimer(IN := (State = 30) AND FiniteMove AND (FaultCode = 0), PT := MoveTimeout);
StopTimer(IN := (State = 40) AND NOT StopTimerStart AND (FaultCode = 0), PT := StopTimeout);

IF FaultCode = 0 THEN
    IF EnableTimer.Q THEN
        FaultCode := 4;
    ELSIF SyncTimer.Q THEN
        FaultCode := 5;
    ELSIF FollowingTimer.Q THEN
        FaultCode := 6;
    ELSIF MoveTimer.Q OR StopTimer.Q THEN
        FaultCode := 7;
    ELSIF SettleTimer.Q THEN
        InTarget := (State = 30) AND FiniteMove;
        State := 20;
        TrajectoryVelocity := 0.0;
        CompletedThisCycle := TRUE;
        FOR I := 1 TO ActiveCount DO
            DriveCommand[I] := 0.0;
        END_FOR;
    END_IF;
END_IF;

//All outputs pass through this final override, including faults detected this scan.
IF (FaultCode <> 0) OR ResetActive OR NOT Commissioned OR Inhibit OR EmergencyStop
    OR RestartBlocked OR NOT ConfigLoaded OR NOT FeedbackInitialized OR NOT HealthyInputs THEN
    TrajectoryVelocity := 0.0;
    FOR I := 1 TO ActiveCount DO
        DriveEnableStep[I] := 0;
        DriveControl[I] := 0;
        DriveCommand[I] := 0.0;
    END_FOR;
    IF ResetActive THEN
        State := 80;
        IF ResetPulse THEN
            DriveControl[1] := 128;
            IF ActiveCount = 2 THEN DriveControl[2] := 128; END_IF;
        END_IF;
    ELSIF FaultCode <> 0 THEN
        State := 90;
        RestartBlocked := TRUE;
        InTarget := FALSE;
    ELSE
        State := 0;
    END_IF;
ELSE
    Busy := (State = 30) OR (State = 40);
    Ready := AllEnabled AND ((State = 20) OR CompletedThisCycle);
    IF AllEnabled AND Busy THEN
        FOR I := 1 TO ActiveCount DO
            RawCommand := DriveCommand[I] / 200.0 * CfgRatio[I]
                * INT_TO_LREAL(CfgDirection[I]) * CfgVelocityUnits[I];
            IF I = 1 THEN
                TargetVelocity1 := LREAL_TO_DINT(RawCommand);
            ELSE
                TargetVelocity2 := LREAL_TO_DINT(RawCommand);
            END_IF;
        END_FOR;
    END_IF;
END_IF;
Controlword1 := DriveControl[1];
IF ActiveCount = 2 THEN
    Controlword2 := DriveControl[2];
ELSE
    DriveControl[2] := 0;
    DriveCommand[2] := 0.0;
    DriveEnableStep[2] := 0;
    Controlword2 := 0;
    TargetVelocity2 := 0;
END_IF;
Error := FaultCode <> 0;
Warning := Warning OR (LimitedSpeed AND Busy);
StmStatus := 0;
IF Ready THEN StmStatus := StmStatus OR WORD#16#0001; END_IF;
IF Busy THEN StmStatus := StmStatus OR WORD#16#0002; END_IF;
IF Error THEN StmStatus := StmStatus OR WORD#16#0008; END_IF;
IF Warning THEN StmStatus := StmStatus OR WORD#16#0080; END_IF;

END_FUNCTION_BLOCK

// ---- POUs/FB_CsvDriveSettings.TcPOU
FUNCTION_BLOCK FB_CsvDriveSettings
VAR_INPUT
    Online : BOOL;
END_VAR
VAR_OUTPUT
    Valid : BOOL;
    ActualMode : USINT;
    ManualBrakeRelease : BOOL;
    ActualTorqueOffset : INT;
    ReadError : BOOL;
    AdsError : UDINT;
END_VAR
VAR
    ReadMode : FB_EcCoeSdoRead;
    ReadBrake : FB_EcCoeSdoRead;
    ReadOffset : FB_EcCoeSdoRead;
    Phase : UINT;
    Trigger : BOOL;
    Completed : BOOL;
    Good : BOOL;
    PollTimer : TON;
    StaleTimer : TON;
END_VAR

//Read-only CoE. Addresses belong to Device 3 Term 7 of the documented machine.
//No mode, brake, limit, reset or other device parameter is written here.
Completed := FALSE;
PollTimer(IN := Phase = 0, PT := T#100MS);
Trigger := (Phase = 0) AND PollTimer.Q AND Online;
ReadMode(sNetId := '10.145.4.14.4.1', nSlaveAddr := 1002,
    nIndex := 16#6010, nSubIndex := 3, pDstBuf := ADR(ActualMode),
    cbBufLen := SIZEOF(ActualMode), bExecute := Trigger, tTimeout := T#200MS);
ReadBrake(sNetId := '10.145.4.14.4.1', nSlaveAddr := 1002,
    nIndex := 16#8012, nSubIndex := 1, pDstBuf := ADR(ManualBrakeRelease),
    cbBufLen := SIZEOF(ManualBrakeRelease), bExecute := Trigger, tTimeout := T#200MS);
ReadOffset(sNetId := '10.145.4.14.4.1', nSlaveAddr := 1002,
    nIndex := 16#7010, nSubIndex := 10, pDstBuf := ADR(ActualTorqueOffset),
    cbBufLen := SIZEOF(ActualTorqueOffset), bExecute := Trigger, tTimeout := T#200MS);
IF Trigger THEN
    Phase := 1;
ELSIF (Phase = 1) AND NOT ReadMode.bBusy AND NOT ReadBrake.bBusy AND NOT ReadOffset.bBusy THEN
    Completed := TRUE;
    ReadError := ReadMode.bError OR ReadBrake.bError OR ReadOffset.bError
        OR (ReadMode.cbRead <> 1) OR (ReadBrake.cbRead <> 1) OR (ReadOffset.cbRead <> 2);
    AdsError := 0;
    IF ReadMode.bError THEN AdsError := ReadMode.nErrId;
    ELSIF ReadBrake.bError THEN AdsError := ReadBrake.nErrId;
    ELSIF ReadOffset.bError THEN AdsError := ReadOffset.nErrId; END_IF;
    Good := NOT ReadError AND (ActualMode = 9) AND NOT ManualBrakeRelease AND (ActualTorqueOffset = 0);
    Phase := 0;
END_IF;
StaleTimer(IN := NOT Completed, PT := T#500MS);
IF NOT Online OR StaleTimer.Q THEN Good := FALSE; END_IF;
Valid := Good AND Online AND NOT StaleTimer.Q AND (ActualMode = 9)
    AND NOT ManualBrakeRelease AND (ActualTorqueOffset = 0);

END_FUNCTION_BLOCK
